QRS_NEXT_CUT()
PTP {E1 28616.845,E2 28616.845}
PTP {X 0,Y 607.911,A -85,B 0,C 180,E1 28616.845,E2 28616.845,E3 0,E4 0,E5 0,E6 0}
QRS_SPEED_INIT()
LIN {X 0,Y 607.911,Z 1007,A -85,B 0,C 180,E1 28616.845,E2 28616.845,E3 0,E4 0,E5 0,E6 0} C_VEL
LIN {X 0,Y 607.911,Z 513.151,A -85,B 0,C 180,E1 28616.845,E2 28616.845} C_VEL
LIN {X 0,Y 607.911,Z 505.074,A -85,B 0,C 180,E1 28616.845,E2 28616.845} C_VEL
LIN {X 0,Y 607.884,Z 503.074,A -85,B 0,C 180,E1 28616.656,E2 28616.656} C_VEL
LIN {X 0,Y 607.844,Z 503.075,A -85,B 0,C 180,E1 28613.767,E2 28613.767} C_VEL
LIN {X 0,Y 607.909,Z 503.072,A -85,B 0,C 180,E1 28610.629,E2 28610.629} C_VEL
LIN {X 0,Y 607.85,Z 503.075,A -85,B 0,C 180,E1 28607.652,E2 28607.652} C_VEL
LIN {X 0,Y 607.919,Z 503.071,A -85,B 0,C 180,E1 28604.516,E2 28604.516} C_VEL
LIN {X 0,Y 607.857,Z 503.074,A -85,B 0,C 180,E1 28601.49,E2 28601.49} C_VEL
LIN {X 0,Y 607.914,Z 503.072,A -85,B 0,C 180,E1 28598.381,E2 28598.381} C_VEL
LIN {X 0,Y 607.861,Z 503.073,A -85,B 0,C 180,E1 28595.408,E2 28595.408} C_VEL
LIN {X 0,Y 607.914,Z 503.074,A -85,B 0,C 180,E1 28592.366,E2 28592.366} C_VEL
LIN {X 0,Y 607.868,Z 503.073,A -85,B 0,C 180,E1 28589.232,E2 28589.232} C_VEL
LIN {X 0,Y 607.912,Z 503.072,A -85,B 0,C 180,E1 28586.112,E2 28586.112} C_VEL
LIN {X 0,Y 607.875,Z 503.073,A -85,B 0,C 180,E1 28582.985,E2 28582.985} C_VEL
LIN {X 0,Y 607.911,Z 503.07,A -85,B 0,C 180,E1 28579.853,E2 28579.853} C_VEL
LIN {X 0,Y 607.88,Z 503.075,A -85,B 0,C 180,E1 28576.767,E2 28576.767} C_VEL
LIN {X 0,Y 607.909,Z 503.417,A -85,B 0,C 180,E1 28576.324,E2 28576.324} C_VEL
LIN {X 0,Y 607.911,Z 532.423,A -85,B 0,C 180,E1 28573.229,E2 28573.229} C_VEL
LIN {X 0,Y 607.861,Z 561.577,A -85,B 0,C 180,E1 28570.197,E2 28570.197} C_VEL
LIN {X 0,Y 607.901,Z 593.601,A -85,B 0,C 180,E1 28566.93,E2 28566.93} C_VEL
LIN {X 0,Y 607.866,Z 623.977,A -85,B 0,C 180,E1 28563.886,E2 28563.886} C_VEL
LIN {X 0,Y 607.91,Z 633.18,A -85,B 0,C 180,E1 28563.011,E2 28563.011} C_VEL
LIN {X 0,Y 607.879,Z 744.156,A -85,B 0,C 180,E1 28561.669,E2 28561.669} C_VEL
LIN {X 0,Y 607.913,Z 759.228,A -85,B 0,C 180,E1 28561.31,E2 28561.31} C_VEL
LIN {X 0,Y 607.919,Z 774.015,A -85,B 0,C 180,E1 28560.76,E2 28560.76} C_VEL
LIN {X 0,Y 607.887,Z 786.969,A -85,B 0,C 180,E1 28560.097,E2 28560.097} C_VEL
LIN {X 0,Y 607.92,Z 799.139,A -85,B 0,C 180,E1 28559.289,E2 28559.289} C_VEL
LIN {X 0,Y 607.919,Z 809.968,A -85,B 0,C 180,E1 28558.366,E2 28558.366} C_VEL
LIN {X 0,Y 607.917,Z 819.55,A -85,B 0,C 180,E1 28557.357,E2 28557.357} C_VEL
LIN {X 0,Y 607.917,Z 828.81,A -85,B 0,C 180,E1 28556.1,E2 28556.1} C_VEL
LIN {X 0,Y 607.917,Z 836.072,A -85,B 0,C 180,E1 28554.784,E2 28554.784} C_VEL
LIN {X 0,Y 607.916,Z 841.374,A -85,B 0,C 180,E1 28553.451,E2 28553.451} C_VEL
LIN {X 0,Y 607.917,Z 845.07,A -85,B 0,C 180,E1 28552.021,E2 28552.021} C_VEL
LIN {X 0,Y 607.918,Z 846.862,A -85,B 0,C 180,E1 28550.504,E2 28550.504} C_VEL
LIN {X 0,Y 607.914,Z 846.58,A -85,B 0,C 180,E1 28549.002,E2 28549.002} C_VEL
LIN {X 0,Y 607.914,Z 844.49,A -85,B 0,C 180,E1 28547.613,E2 28547.613} C_VEL
LIN {X 0,Y 607.915,Z 840.63,A -85,B 0,C 180,E1 28546.234,E2 28546.234} C_VEL
LIN {X 0,Y 607.915,Z 834.801,A -85,B 0,C 180,E1 28544.865,E2 28544.865} C_VEL
LIN {X 0,Y 607.915,Z 827.41,A -85,B 0,C 180,E1 28543.601,E2 28543.601} C_VEL
LIN {X 0,Y 607.919,Z 818.592,A -85,B 0,C 180,E1 28542.44,E2 28542.44} C_VEL
LIN {X 0,Y 607.918,Z 807.23,A -85,B 0,C 180,E1 28541.285,E2 28541.285} C_VEL
LIN {X 0,Y 607.915,Z 795.047,A -85,B 0,C 180,E1 28540.326,E2 28540.326} C_VEL
LIN {X 0,Y 607.906,Z 781.548,A -85,B 0,C 180,E1 28539.513,E2 28539.513} C_VEL
LIN {X 0,Y 607.917,Z 767.716,A -85,B 0,C 180,E1 28538.892,E2 28538.892} C_VEL
LIN {X 0,Y 607.918,Z 753.447,A -85,B 0,C 180,E1 28538.439,E2 28538.439} C_VEL
LIN {X 0,Y 607.905,Z 737.614,A -85,B 0,C 180,E1 28538.142,E2 28538.142} C_VEL
LIN {X 0,Y 607.918,Z 633.091,A -85,B 0,C 180,E1 28536.894,E2 28536.894} C_VEL
LIN {X 0,Y 607.891,Z 611.812,A -85,B 0,C 180,E1 28534.81,E2 28534.81} C_VEL
LIN {X 0,Y 607.883,Z 580.938,A -85,B 0,C 180,E1 28531.695,E2 28531.695} C_VEL
LIN {X 0,Y 607.916,Z 551.557,A -85,B 0,C 180,E1 28528.68,E2 28528.68} C_VEL
LIN {X 0,Y 607.916,Z 520.967,A -85,B 0,C 180,E1 28525.471,E2 28525.471} C_VEL
LIN {X 0,Y 607.9,Z 503.204,A -85,B 0,C 180,E1 28523.542,E2 28523.542} C_VEL
LIN {X 0,Y 607.833,Z 503.077,A -85,B 0,C 180,E1 28520.627,E2 28520.627} C_VEL
LIN {X 0,Y 607.908,Z 503.075,A -85,B 0,C 180,E1 28517.654,E2 28517.654} C_VEL
LIN {X 0,Y 607.83,Z 503.077,A -85,B 0,C 180,E1 28514.545,E2 28514.545} C_VEL
LIN {X 0,Y 607.871,Z 503.076,A -85,B 0,C 180,E1 28511.69,E2 28511.69} C_VEL
LIN {X 0,Y 607.837,Z 503.077,A -85,B 0,C 180,E1 28508.582,E2 28508.582} C_VEL
LIN {X 0,Y 607.837,Z 503.076,A -85,B 0,C 180,E1 28505.822,E2 28505.822} C_VEL
LIN {X 0,Y 607.848,Z 503.077,A -85,B 0,C 180,E1 28502.577,E2 28502.577} C_VEL
LIN {X 0,Y 607.826,Z 503.076,A -85,B 0,C 180,E1 28499.779,E2 28499.779} C_VEL
LIN {X 0,Y 607.882,Z 503.077,A -85,B 0,C 180,E1 28496.676,E2 28496.676} C_VEL
LIN {X 0,Y 607.824,Z 503.077,A -85,B 0,C 180,E1 28493.806,E2 28493.806} C_VEL
LIN {X 0,Y 607.913,Z 503.078,A -85,B 0,C 180,E1 28490.714,E2 28490.714} C_VEL
LIN {X 0,Y 607.828,Z 503.076,A -85,B 0,C 180,E1 28487.72,E2 28487.72} C_VEL
LIN {X 0,Y 607.858,Z 503.077,A -85,B 0,C 180,E1 28484.988,E2 28484.988} C_VEL
LIN {X 0,Y 607.841,Z 503.076,A -85,B 0,C 180,E1 28481.775,E2 28481.775} C_VEL
LIN {X 0,Y 607.841,Z 503.076,A -85,B 0,C 180,E1 28479.051,E2 28479.051} C_VEL
LIN {X 0,Y 607.864,Z 503.075,A -85,B 0,C 180,E1 28475.819,E2 28475.819} C_VEL
LIN {X 0,Y 607.835,Z 503.076,A -85,B 0,C 180,E1 28473.102,E2 28473.102} C_VEL
LIN {X 0,Y 607.918,Z 503.074,A -85,B 0,C 180,E1 28470,E2 28470} C_VEL
LIN {X 0,Y 607.837,Z 503.075,A -85,B 0,C 180,E1 28467.001,E2 28467.001} C_VEL
LIN {X 0,Y 607.917,Z 503.077,A -85,B 0,C 180,E1 28463.97,E2 28463.97} C_VEL
LIN {X 0,Y 607.841,Z 503.075,A -85,B 0,C 180,E1 28460.891,E2 28460.891} C_VEL
LIN {X 0,Y 607.904,Z 503.077,A -85,B 0,C 180,E1 28457.913,E2 28457.913} C_VEL
LIN {X 0,Y 607.85,Z 503.074,A -85,B 0,C 180,E1 28454.869,E2 28454.869} C_VEL
LIN {X 0,Y 607.876,Z 503.076,A -85,B 0,C 180,E1 28451.961,E2 28451.961} C_VEL
LIN {X 0,Y 607.86,Z 503.073,A -85,B 0,C 180,E1 28448.8,E2 28448.8} C_VEL
LIN {X 0,Y 607.863,Z 503.076,A -85,B 0,C 180,E1 28445.948,E2 28445.948} C_VEL
LIN {X 0,Y 607.865,Z 503.073,A -85,B 0,C 180,E1 28442.64,E2 28442.64} C_VEL
LIN {X 0,Y 607.869,Z 503.075,A -85,B 0,C 180,E1 28439.717,E2 28439.717} C_VEL
LIN {X 0,Y 607.865,Z 503.072,A -85,B 0,C 180,E1 28436.417,E2 28436.417} C_VEL
LIN {X 0,Y 607.876,Z 503.076,A -85,B 0,C 180,E1 28433.483,E2 28433.483} C_VEL
LIN {X 0,Y 607.869,Z 503.072,A -85,B 0,C 180,E1 28430.246,E2 28430.246} C_VEL
LIN {X 0,Y 607.883,Z 503.076,A -85,B 0,C 180,E1 28427.242,E2 28427.242} C_VEL
LIN {X 0,Y 607.872,Z 503.071,A -85,B 0,C 180,E1 28424.057,E2 28424.057} C_VEL
LIN {X 0,Y 607.888,Z 503.076,A -85,B 0,C 180,E1 28421.032,E2 28421.032} C_VEL
LIN {X 0,Y 607.868,Z 503.072,A -85,B 0,C 180,E1 28417.771,E2 28417.771} C_VEL
LIN {X 0,Y 607.899,Z 503.077,A -85,B 0,C 180,E1 28414.765,E2 28414.765} C_VEL
LIN {X 0,Y 607.872,Z 503.071,A -85,B 0,C 180,E1 28411.617,E2 28411.617} C_VEL
LIN {X 0,Y 607.902,Z 503.077,A -85,B 0,C 180,E1 28408.574,E2 28408.574} C_VEL
LIN {X 0,Y 607.873,Z 503.071,A -85,B 0,C 180,E1 28405.426,E2 28405.426} C_VEL
LIN {X 0,Y 607.914,Z 503.078,A -85,B 0,C 180,E1 28402.286,E2 28402.286} C_VEL
LIN {X 0,Y 607.871,Z 503.071,A -85,B 0,C 180,E1 28399.107,E2 28399.107} C_VEL
LIN {X 0,Y 607.914,Z 503.075,A -85,B 0,C 180,E1 28395.948,E2 28395.948} C_VEL
LIN {X 0,Y 607.87,Z 503.072,A -85,B 0,C 180,E1 28392.811,E2 28392.811} C_VEL
LIN {X 0,Y 607.914,Z 503.075,A -85,B 0,C 180,E1 28389.774,E2 28389.774} C_VEL
LIN {X 0,Y 607.873,Z 503.072,A -85,B 0,C 180,E1 28386.613,E2 28386.613} C_VEL
LIN {X 0,Y 607.911,Z 503.073,A -85,B 0,C 180,E1 28383.5,E2 28383.5} C_VEL
LIN {X 0,Y 607.875,Z 503.072,A -85,B 0,C 180,E1 28380.437,E2 28380.437} C_VEL
LIN {X 0,Y 607.901,Z 503.299,A -85,B 0,C 180,E1 28379.782,E2 28379.782} C_VEL
LIN {X 0,Y 607.917,Z 514.846,A -85,B 0,C 180,E1 28378.956,E2 28378.956} C_VEL
LIN {X 0,Y 607.891,Z 559.528,A -85,B 0,C 180,E1 28375.944,E2 28375.944} C_VEL
LIN {X 0,Y 607.91,Z 607.569,A -85,B 0,C 180,E1 28372.788,E2 28372.788} C_VEL
LIN {X 0,Y 607.906,Z 615.06,A -85,B 0,C 180,E1 28372.329,E2 28372.329} C_VEL
LIN {X 0,Y 607.912,Z 824.351,A -85,B 0,C 180,E1 28369.704,E2 28369.704} C_VEL
LIN {X 0,Y 607.892,Z 842.612,A -85,B 0,C 180,E1 28369.305,E2 28369.305} C_VEL
LIN {X 0,Y 607.91,Z 860.78,A -85,B 0,C 180,E1 28368.731,E2 28368.731} C_VEL
LIN {X 0,Y 607.886,Z 879.07,A -85,B 0,C 180,E1 28367.963,E2 28367.963} C_VEL
LIN {X 0,Y 607.919,Z 895.797,A -85,B 0,C 180,E1 28367.072,E2 28367.072} C_VEL
LIN {X 0,Y 607.916,Z 911.646,A -85,B 0,C 180,E1 28366.04,E2 28366.04} C_VEL
LIN {X 0,Y 607.917,Z 926.565,A -85,B 0,C 180,E1 28364.867,E2 28364.867} C_VEL
LIN {X 0,Y 607.918,Z 940.218,A -85,B 0,C 180,E1 28363.582,E2 28363.582} C_VEL
LIN {X 0,Y 607.917,Z 952.906,A -85,B 0,C 180,E1 28362.153,E2 28362.153} C_VEL
LIN {X 0,Y 607.913,Z 964.223,A -85,B 0,C 180,E1 28360.615,E2 28360.615} C_VEL
LIN {X 0,Y 607.918,Z 973.987,A -85,B 0,C 180,E1 28358.99,E2 28358.99} C_VEL
LIN {X 0,Y 607.909,Z 981.864,A -85,B 0,C 180,E1 28357.35,E2 28357.35} C_VEL
LIN {X 0,Y 607.906,Z 988.106,A -85,B 0,C 180,E1 28355.664,E2 28355.664} C_VEL
LIN {X 0,Y 607.917,Z 992.871,A -85,B 0,C 180,E1 28353.867,E2 28353.867} C_VEL
LIN {X 0,Y 607.916,Z 995.786,A -85,B 0,C 180,E1 28352.075,E2 28352.075} C_VEL
LIN {X 0,Y 607.907,Z 996.939,A -85,B 0,C 180,E1 28350.284,E2 28350.284} C_VEL
LIN {X 0,Y 607.915,Z 996.349,A -85,B 0,C 180,E1 28348.493,E2 28348.493} C_VEL
LIN {X 0,Y 607.908,Z 994.007,A -85,B 0,C 180,E1 28346.701,E2 28346.701} C_VEL
LIN {X 0,Y 607.905,Z 990.1,A -85,B 0,C 180,E1 28345.001,E2 28345.001} C_VEL
LIN {X 0,Y 607.913,Z 984.473,A -85,B 0,C 180,E1 28343.296,E2 28343.296} C_VEL
LIN {X 0,Y 607.915,Z 977.431,A -85,B 0,C 180,E1 28341.68,E2 28341.68} C_VEL
LIN {X 0,Y 607.91,Z 968.521,A -85,B 0,C 180,E1 28340.057,E2 28340.057} C_VEL
LIN {X 0,Y 607.919,Z 958.16,A -85,B 0,C 180,E1 28338.523,E2 28338.523} C_VEL
LIN {X 0,Y 607.914,Z 946.365,A -85,B 0,C 180,E1 28337.077,E2 28337.077} C_VEL
LIN {X 0,Y 607.916,Z 933.113,A -85,B 0,C 180,E1 28335.72,E2 28335.72} C_VEL
LIN {X 0,Y 607.917,Z 918.266,A -85,B 0,C 180,E1 28334.452,E2 28334.452} C_VEL
LIN {X 0,Y 607.918,Z 902.26,A -85,B 0,C 180,E1 28333.324,E2 28333.324} C_VEL
LIN {X 0,Y 607.895,Z 886.08,A -85,B 0,C 180,E1 28332.386,E2 28332.386} C_VEL
LIN {X 0,Y 607.907,Z 869.132,A -85,B 0,C 180,E1 28331.594,E2 28331.594} C_VEL
LIN {X 0,Y 607.892,Z 850.474,A -85,B 0,C 180,E1 28330.922,E2 28330.922} C_VEL
LIN {X 0,Y 607.901,Z 832.403,A -85,B 0,C 180,E1 28330.451,E2 28330.451} C_VEL
LIN {X 0,Y 607.919,Z 812.939,A -85,B 0,C 180,E1 28330.13,E2 28330.13} C_VEL
LIN {X 0,Y 607.906,Z 614.386,A -85,B 0,C 180,E1 28327.648,E2 28327.648} C_VEL
LIN {X 0,Y 607.907,Z 568.229,A -85,B 0,C 180,E1 28324.634,E2 28324.634} C_VEL
LIN {X 0,Y 607.917,Z 521.763,A -85,B 0,C 180,E1 28321.516,E2 28321.516} C_VEL
LIN {X 0,Y 607.904,Z 503.513,A -85,B 0,C 180,E1 28320.249,E2 28320.249} C_VEL
LIN {X 0,Y 607.883,Z 503.075,A -85,B 0,C 180,E1 28320.003,E2 28320.003} C_VEL
LIN {X 0,Y 607.917,Z 503.068,A -85,B 0,C 180,E1 28316.842,E2 28316.842} C_VEL
LIN {X 0,Y 607.873,Z 503.074,A -85,B 0,C 180,E1 28313.696,E2 28313.696} C_VEL
LIN {X 0,Y 607.915,Z 503.07,A -85,B 0,C 180,E1 28310.595,E2 28310.595} C_VEL
LIN {X 0,Y 607.864,Z 503.074,A -85,B 0,C 180,E1 28307.468,E2 28307.468} C_VEL
LIN {X 0,Y 607.918,Z 503.07,A -85,B 0,C 180,E1 28304.461,E2 28304.461} C_VEL
LIN {X 0,Y 607.858,Z 503.074,A -85,B 0,C 180,E1 28301.268,E2 28301.268} C_VEL
LIN {X 0,Y 607.918,Z 503.072,A -85,B 0,C 180,E1 28298.178,E2 28298.178} C_VEL
LIN {X 0,Y 607.852,Z 503.075,A -85,B 0,C 180,E1 28295.15,E2 28295.15} C_VEL
LIN {X 0,Y 607.91,Z 503.072,A -85,B 0,C 180,E1 28292.118,E2 28292.118} C_VEL
LIN {X 0,Y 607.847,Z 503.075,A -85,B 0,C 180,E1 28289.029,E2 28289.029} C_VEL
LIN {X 0,Y 607.883,Z 503.074,A -85,B 0,C 180,E1 28286.107,E2 28286.107} C_VEL
LIN {X 0,Y 607.842,Z 503.076,A -85,B 0,C 180,E1 28282.918,E2 28282.918} C_VEL
LIN {X 0,Y 607.859,Z 503.075,A -85,B 0,C 180,E1 28280.095,E2 28280.095} C_VEL
LIN {X 0,Y 607.839,Z 503.077,A -85,B 0,C 180,E1 28276.828,E2 28276.828} C_VEL
LIN {X 0,Y 607.833,Z 503.076,A -85,B 0,C 180,E1 28274.188,E2 28274.188} C_VEL
LIN {X 0,Y 607.862,Z 503.077,A -85,B 0,C 180,E1 28271,E2 28271} C_VEL
LIN {X 0,Y 607.825,Z 503.077,A -85,B 0,C 180,E1 28268.228,E2 28268.228} C_VEL
LIN {X 0,Y 607.913,Z 503.077,A -85,B 0,C 180,E1 28265.19,E2 28265.19} C_VEL
LIN {X 0,Y 607.833,Z 503.076,A -85,B 0,C 180,E1 28262.168,E2 28262.168} C_VEL
LIN {X 0,Y 607.909,Z 503.078,A -85,B 0,C 180,E1 28259.152,E2 28259.152} C_VEL
LIN {X 0,Y 607.884,Z 503.074,A -85,B 0,C 180,E1 28256.656,E2 28256.656} C_VEL
LIN {X 0,Y 606.826,Z 503.205,A -85,B 0,C 180,E1 28255.93,E2 28255.93} C_VEL
LIN {X 0,Y 600.415,Z 504.003,A -85,B 0,C 180,E1 28253.894,E2 28253.894} C_VEL
LIN {X 0,Y 599.932,Z 504.065,A -85,B 0,C 180,E1 28253.364,E2 28253.364} C_VEL
LIN {X 0,Y 599.917,Z 504.062,A -85,B 0,C 180,E1 28250.115,E2 28250.115} C_VEL
LIN {X 0,Y 599.939,Z 504.065,A -85,B 0,C 180,E1 28247.193,E2 28247.193} C_VEL
LIN {X 0,Y 599.923,Z 504.062,A -85,B 0,C 180,E1 28243.939,E2 28243.939} C_VEL
LIN {X 0,Y 599.963,Z 504.066,A -85,B 0,C 180,E1 28240.878,E2 28240.878} C_VEL
LIN {X 0,Y 599.924,Z 504.062,A -85,B 0,C 180,E1 28237.651,E2 28237.651} C_VEL
LIN {X 0,Y 599.978,Z 504.065,A -85,B 0,C 180,E1 28234.535,E2 28234.535} C_VEL
LIN {X 0,Y 599.928,Z 504.062,A -85,B 0,C 180,E1 28231.424,E2 28231.424} C_VEL
LIN {X 0,Y 599.976,Z 504.064,A -85,B 0,C 180,E1 28228.335,E2 28228.335} C_VEL
LIN {X 0,Y 599.934,Z 504.061,A -85,B 0,C 180,E1 28225.24,E2 28225.24} C_VEL
LIN {X 0,Y 599.974,Z 504.064,A -85,B 0,C 180,E1 28222.17,E2 28222.17} C_VEL
LIN {X 0,Y 599.939,Z 504.063,A -85,B 0,C 180,E1 28218.955,E2 28218.955} C_VEL
LIN {X 0,Y 599.983,Z 504.317,A -85,B 0,C 180,E1 28216.609,E2 28216.609} C_VEL
LIN {X 0,Y 600.305,Z 508.323,A -85,B 0,C 180,E1 28216.141,E2 28216.141} C_VEL
LIN {X 0,Y 600.213,Z 538.089,A -85,B 0,C 180,E1 28212.941,E2 28212.941} C_VEL
LIN {X 0,Y 600.13,Z 568.295,A -85,B 0,C 180,E1 28209.769,E2 28209.769} C_VEL
LIN {X 0,Y 600.067,Z 599.365,A -85,B 0,C 180,E1 28206.569,E2 28206.569} C_VEL
LIN {X 0,Y 600.003,Z 631.076,A -85,B 0,C 180,E1 28203.357,E2 28203.357} C_VEL
LIN {X 0,Y 600.096,Z 633.638,A -85,B 0,C 180,E1 28203.176,E2 28203.176} C_VEL
LIN {X 0,Y 600.042,Z 744.434,A -85,B 0,C 180,E1 28201.819,E2 28201.819} C_VEL
LIN {X 0,Y 600.058,Z 759.369,A -85,B 0,C 180,E1 28201.456,E2 28201.456} C_VEL
LIN {X 0,Y 600.039,Z 774.355,A -85,B 0,C 180,E1 28200.889,E2 28200.889} C_VEL
LIN {X 0,Y 599.979,Z 787.292,A -85,B 0,C 180,E1 28200.213,E2 28200.213} C_VEL
LIN {X 0,Y 599.985,Z 799.854,A -85,B 0,C 180,E1 28199.358,E2 28199.358} C_VEL
LIN {X 0,Y 599.962,Z 810.146,A -85,B 0,C 180,E1 28198.461,E2 28198.461} C_VEL
LIN {X 0,Y 599.943,Z 819.714,A -85,B 0,C 180,E1 28197.436,E2 28197.436} C_VEL
LIN {X 0,Y 599.931,Z 828.658,A -85,B 0,C 180,E1 28196.206,E2 28196.206} C_VEL
LIN {X 0,Y 599.923,Z 835.651,A -85,B 0,C 180,E1 28194.936,E2 28194.936} C_VEL
LIN {X 0,Y 599.92,Z 840.797,A -85,B 0,C 180,E1 28193.679,E2 28193.679} C_VEL
LIN {X 0,Y 599.916,Z 844.706,A -85,B 0,C 180,E1 28192.227,E2 28192.227} C_VEL
LIN {X 0,Y 599.915,Z 846.599,A -85,B 0,C 180,E1 28190.892,E2 28190.892} C_VEL
LIN {X 0,Y 599.915,Z 846.893,A -85,B 0,C 180,E1 28189.468,E2 28189.468} C_VEL
LIN {X 0,Y 599.917,Z 845.391,A -85,B 0,C 180,E1 28188.056,E2 28188.056} C_VEL
LIN {X 0,Y 599.917,Z 842.141,A -85,B 0,C 180,E1 28186.656,E2 28186.656} C_VEL
LIN {X 0,Y 599.92,Z 836.744,A -85,B 0,C 180,E1 28185.204,E2 28185.204} C_VEL
LIN {X 0,Y 599.929,Z 829.752,A -85,B 0,C 180,E1 28183.884,E2 28183.884} C_VEL
LIN {X 0,Y 599.942,Z 821.575,A -85,B 0,C 180,E1 28182.706,E2 28182.706} C_VEL
LIN {X 0,Y 599.958,Z 812.955,A -85,B 0,C 180,E1 28181.729,E2 28181.729} C_VEL
LIN {X 0,Y 599.979,Z 802.998,A -85,B 0,C 180,E1 28180.804,E2 28180.804} C_VEL
LIN {X 0,Y 599.984,Z 790.324,A -85,B 0,C 180,E1 28179.882,E2 28179.882} C_VEL
LIN {X 0,Y 600.029,Z 777.198,A -85,B 0,C 180,E1 28179.155,E2 28179.155} C_VEL
LIN {X 0,Y 600.057,Z 763.751,A -85,B 0,C 180,E1 28178.598,E2 28178.598} C_VEL
LIN {X 0,Y 600.076,Z 748.239,A -85,B 0,C 180,E1 28178.164,E2 28178.164} C_VEL
LIN {X 0,Y 600.068,Z 729.544,A -85,B 0,C 180,E1 28177.887,E2 28177.887} C_VEL
LIN {X 0,Y 600.054,Z 633.14,A -85,B 0,C 180,E1 28176.723,E2 28176.723} C_VEL
LIN {X 0,Y 600.026,Z 620.12,A -85,B 0,C 180,E1 28175.449,E2 28175.449} C_VEL
LIN {X 0,Y 600.054,Z 590.046,A -85,B 0,C 180,E1 28172.386,E2 28172.386} C_VEL
LIN {X 0,Y 600.127,Z 559.615,A -85,B 0,C 180,E1 28169.235,E2 28169.235} C_VEL
LIN {X 0,Y 600.211,Z 530.678,A -85,B 0,C 180,E1 28166.178,E2 28166.178} C_VEL
LIN {X 0,Y 600.23,Z 505.406,A -85,B 0,C 180,E1 28163.447,E2 28163.447} C_VEL
LIN {X 0,Y 599.936,Z 504.157,A -85,B 0,C 180,E1 28163.252,E2 28163.252} C_VEL
LIN {X 0,Y 599.898,Z 504.066,A -85,B 0,C 180,E1 28160.405,E2 28160.405} C_VEL
LIN {X 0,Y 599.949,Z 504.066,A -85,B 0,C 180,E1 28157.292,E2 28157.292} C_VEL
LIN {X 0,Y 599.891,Z 504.066,A -85,B 0,C 180,E1 28154.335,E2 28154.335} C_VEL
LIN {X 0,Y 599.967,Z 504.066,A -85,B 0,C 180,E1 28151.238,E2 28151.238} C_VEL
LIN {X 0,Y 599.888,Z 504.066,A -85,B 0,C 180,E1 28148.284,E2 28148.284} C_VEL
LIN {X 0,Y 599.958,Z 504.063,A -85,B 0,C 180,E1 28145.268,E2 28145.268} C_VEL
LIN {X 0,Y 599.886,Z 504.066,A -85,B 0,C 180,E1 28142.182,E2 28142.182} C_VEL
LIN {X 0,Y 599.937,Z 504.064,A -85,B 0,C 180,E1 28139.228,E2 28139.228} C_VEL
LIN {X 0,Y 599.887,Z 504.066,A -85,B 0,C 180,E1 28136.06,E2 28136.06} C_VEL
LIN {X 0,Y 599.914,Z 504.066,A -85,B 0,C 180,E1 28133.252,E2 28133.252} C_VEL
LIN {X 0,Y 599.901,Z 504.066,A -85,B 0,C 180,E1 28130.058,E2 28130.058} C_VEL
LIN {X 0,Y 599.898,Z 504.065,A -85,B 0,C 180,E1 28127.288,E2 28127.288} C_VEL
LIN {X 0,Y 599.915,Z 504.065,A -85,B 0,C 180,E1 28124.028,E2 28124.028} C_VEL
LIN {X 0,Y 599.898,Z 504.064,A -85,B 0,C 180,E1 28121.175,E2 28121.175} C_VEL
LIN {X 0,Y 599.935,Z 504.064,A -85,B 0,C 180,E1 28117.977,E2 28117.977} C_VEL
LIN {X 0,Y 599.897,Z 504.064,A -85,B 0,C 180,E1 28115.084,E2 28115.084} C_VEL
LIN {X 0,Y 599.966,Z 504.063,A -85,B 0,C 180,E1 28111.983,E2 28111.983} C_VEL
LIN {X 0,Y 599.898,Z 504.065,A -85,B 0,C 180,E1 28108.959,E2 28108.959} C_VEL
LIN {X 0,Y 599.975,Z 504.062,A -85,B 0,C 180,E1 28105.861,E2 28105.861} C_VEL
LIN {X 0,Y 599.901,Z 504.064,A -85,B 0,C 180,E1 28102.835,E2 28102.835} C_VEL
LIN {X 0,Y 599.978,Z 504.063,A -85,B 0,C 180,E1 28099.773,E2 28099.773} C_VEL
LIN {X 0,Y 599.904,Z 504.062,A -85,B 0,C 180,E1 28096.759,E2 28096.759} C_VEL
LIN {X 0,Y 599.966,Z 504.066,A -85,B 0,C 180,E1 28093.787,E2 28093.787} C_VEL
LIN {X 0,Y 599.909,Z 504.062,A -85,B 0,C 180,E1 28090.661,E2 28090.661} C_VEL
LIN {X 0,Y 599.958,Z 504.064,A -85,B 0,C 180,E1 28087.662,E2 28087.662} C_VEL
LIN {X 0,Y 599.913,Z 504.063,A -85,B 0,C 180,E1 28084.493,E2 28084.493} C_VEL
LIN {X 0,Y 599.955,Z 504.065,A -85,B 0,C 180,E1 28081.528,E2 28081.528} C_VEL
LIN {X 0,Y 599.919,Z 504.062,A -85,B 0,C 180,E1 28078.377,E2 28078.377} C_VEL
LIN {X 0,Y 599.948,Z 504.066,A -85,B 0,C 180,E1 28075.412,E2 28075.412} C_VEL
LIN {X 0,Y 599.925,Z 504.06,A -85,B 0,C 180,E1 28072.242,E2 28072.242} C_VEL
LIN {X 0,Y 599.95,Z 504.065,A -85,B 0,C 180,E1 28069.242,E2 28069.242} C_VEL
LIN {X 0,Y 599.926,Z 504.06,A -85,B 0,C 180,E1 28066.015,E2 28066.015} C_VEL
LIN {X 0,Y 599.954,Z 504.065,A -85,B 0,C 180,E1 28063.043,E2 28063.043} C_VEL
LIN {X 0,Y 599.928,Z 504.06,A -85,B 0,C 180,E1 28059.819,E2 28059.819} C_VEL
LIN {X 0,Y 599.978,Z 504.066,A -85,B 0,C 180,E1 28056.661,E2 28056.661} C_VEL
LIN {X 0,Y 599.925,Z 504.06,A -85,B 0,C 180,E1 28053.471,E2 28053.471} C_VEL
LIN {X 0,Y 599.979,Z 504.065,A -85,B 0,C 180,E1 28050.441,E2 28050.441} C_VEL
LIN {X 0,Y 599.928,Z 504.061,A -85,B 0,C 180,E1 28047.309,E2 28047.309} C_VEL
LIN {X 0,Y 599.977,Z 504.064,A -85,B 0,C 180,E1 28044.201,E2 28044.201} C_VEL
LIN {X 0,Y 599.929,Z 504.061,A -85,B 0,C 180,E1 28041.074,E2 28041.074} C_VEL
LIN {X 0,Y 599.974,Z 504.063,A -85,B 0,C 180,E1 28037.938,E2 28037.938} C_VEL
LIN {X 0,Y 599.931,Z 504.061,A -85,B 0,C 180,E1 28034.825,E2 28034.825} C_VEL
LIN {X 0,Y 599.973,Z 504.062,A -85,B 0,C 180,E1 28031.704,E2 28031.704} C_VEL
LIN {X 0,Y 599.933,Z 504.062,A -85,B 0,C 180,E1 28028.556,E2 28028.556} C_VEL
LIN {X 0,Y 599.973,Z 504.061,A -85,B 0,C 180,E1 28025.42,E2 28025.42} C_VEL
LIN {X 0,Y 599.937,Z 504.061,A -85,B 0,C 180,E1 28022.228,E2 28022.228} C_VEL
LIN {X 0,Y 599.972,Z 504.303,A -85,B 0,C 180,E1 28020.143,E2 28020.143} C_VEL
LIN {X 0,Y 600.653,Z 507.548,A -85,B 0,C 180,E1 28019.848,E2 28019.848} C_VEL
LIN {X 0,Y 600.489,Z 551.772,A -85,B 0,C 180,E1 28016.814,E2 28016.814} C_VEL
LIN {X 0,Y 600.375,Z 597.331,A -85,B 0,C 180,E1 28013.766,E2 28013.766} C_VEL
LIN {X 0,Y 600.405,Z 615.06,A -85,B 0,C 180,E1 28012.623,E2 28012.623} C_VEL
LIN {X 0,Y 600.372,Z 824.351,A -85,B 0,C 180,E1 28009.962,E2 28009.962} C_VEL
LIN {X 0,Y 600.312,Z 843.223,A -85,B 0,C 180,E1 28009.541,E2 28009.541} C_VEL
LIN {X 0,Y 600.281,Z 861.422,A -85,B 0,C 180,E1 28008.953,E2 28008.953} C_VEL
LIN {X 0,Y 600.204,Z 879.067,A -85,B 0,C 180,E1 28008.2,E2 28008.2} C_VEL
LIN {X 0,Y 600.179,Z 895.713,A -85,B 0,C 180,E1 28007.304,E2 28007.304} C_VEL
LIN {X 0,Y 600.122,Z 911.645,A -85,B 0,C 180,E1 28006.254,E2 28006.254} C_VEL
LIN {X 0,Y 600.069,Z 926.566,A -85,B 0,C 180,E1 28005.066,E2 28005.066} C_VEL
LIN {X 0,Y 600.02,Z 940.02,A -85,B 0,C 180,E1 28003.786,E2 28003.786} C_VEL
LIN {X 0,Y 599.985,Z 952.907,A -85,B 0,C 180,E1 28002.316,E2 28002.316} C_VEL
LIN {X 0,Y 599.954,Z 964.224,A -85,B 0,C 180,E1 28000.758,E2 28000.758} C_VEL
LIN {X 0,Y 599.934,Z 973.988,A -85,B 0,C 180,E1 27999.11,E2 27999.11} C_VEL
LIN {X 0,Y 599.92,Z 982.043,A -85,B 0,C 180,E1 27997.405,E2 27997.405} C_VEL
LIN {X 0,Y 599.911,Z 988.408,A -85,B 0,C 180,E1 27995.644,E2 27995.644} C_VEL
LIN {X 0,Y 599.918,Z 992.871,A -85,B 0,C 180,E1 27993.919,E2 27993.919} C_VEL
LIN {X 0,Y 599.917,Z 995.786,A -85,B 0,C 180,E1 27992.102,E2 27992.102} C_VEL
LIN {X 0,Y 599.907,Z 996.939,A -85,B 0,C 180,E1 27990.288,E2 27990.288} C_VEL
LIN {X 0,Y 599.915,Z 996.349,A -85,B 0,C 180,E1 27988.473,E2 27988.473} C_VEL
LIN {X 0,Y 599.907,Z 994.008,A -85,B 0,C 180,E1 27986.657,E2 27986.657} C_VEL
LIN {X 0,Y 599.908,Z 990.101,A -85,B 0,C 180,E1 27984.934,E2 27984.934} C_VEL
LIN {X 0,Y 599.92,Z 984.474,A -85,B 0,C 180,E1 27983.206,E2 27983.206} C_VEL
LIN {X 0,Y 599.928,Z 977.432,A -85,B 0,C 180,E1 27981.568,E2 27981.568} C_VEL
LIN {X 0,Y 599.942,Z 968.522,A -85,B 0,C 180,E1 27979.924,E2 27979.924} C_VEL
LIN {X 0,Y 599.969,Z 958.161,A -85,B 0,C 180,E1 27978.369,E2 27978.369} C_VEL
LIN {X 0,Y 600.001,Z 946.366,A -85,B 0,C 180,E1 27976.903,E2 27976.903} C_VEL
LIN {X 0,Y 600.049,Z 932.752,A -85,B 0,C 180,E1 27975.493,E2 27975.493} C_VEL
LIN {X 0,Y 600.103,Z 918.265,A -85,B 0,C 180,E1 27974.244,E2 27974.244} C_VEL
LIN {X 0,Y 600.164,Z 902.263,A -85,B 0,C 180,E1 27973.102,E2 27973.102} C_VEL
LIN {X 0,Y 600.195,Z 885.088,A -85,B 0,C 180,E1 27972.103,E2 27972.103} C_VEL
LIN {X 0,Y 600.277,Z 867.704,A -85,B 0,C 180,E1 27971.295,E2 27971.295} C_VEL
LIN {X 0,Y 600.302,Z 849.613,A -85,B 0,C 180,E1 27970.646,E2 27970.646} C_VEL
LIN {X 0,Y 600.354,Z 831.296,A -85,B 0,C 180,E1 27970.173,E2 27970.173} C_VEL
LIN {X 0,Y 600.395,Z 811.501,A -85,B 0,C 180,E1 27969.852,E2 27969.852} C_VEL
LIN {X 0,Y 600.379,Z 614.841,A -85,B 0,C 180,E1 27967.371,E2 27967.371} C_VEL
LIN {X 0,Y 600.463,Z 568.229,A -85,B 0,C 180,E1 27964.297,E2 27964.297} C_VEL
LIN {X 0,Y 600.607,Z 521.554,A -85,B 0,C 180,E1 27961.123,E2 27961.123} C_VEL
LIN {X 0,Y 600.44,Z 506.011,A -85,B 0,C 180,E1 27960.033,E2 27960.033} C_VEL
LIN {X 0,Y 599.951,Z 504.171,A -85,B 0,C 180,E1 27959.816,E2 27959.816} C_VEL
LIN {X 0,Y 599.975,Z 504.059,A -85,B 0,C 180,E1 27956.756,E2 27956.756} C_VEL
LIN {X 0,Y 599.932,Z 504.063,A -85,B 0,C 180,E1 27953.608,E2 27953.608} C_VEL
LIN {X 0,Y 599.975,Z 504.061,A -85,B 0,C 180,E1 27950.467,E2 27950.467} C_VEL
LIN {X 0,Y 599.925,Z 504.063,A -85,B 0,C 180,E1 27947.423,E2 27947.423} C_VEL
LIN {X 0,Y 599.977,Z 504.06,A -85,B 0,C 180,E1 27944.37,E2 27944.37} C_VEL
LIN {X 0,Y 599.92,Z 504.063,A -85,B 0,C 180,E1 27941.273,E2 27941.273} C_VEL
LIN {X 0,Y 599.978,Z 504.061,A -85,B 0,C 180,E1 27938.141,E2 27938.141} C_VEL
LIN {X 0,Y 599.912,Z 504.063,A -85,B 0,C 180,E1 27935.09,E2 27935.09} C_VEL
LIN {X 0,Y 599.979,Z 504.062,A -85,B 0,C 180,E1 27931.989,E2 27931.989} C_VEL
LIN {X 0,Y 599.905,Z 504.064,A -85,B 0,C 180,E1 27928.904,E2 27928.904} C_VEL
LIN {X 0,Y 599.973,Z 504.063,A -85,B 0,C 180,E1 27925.866,E2 27925.866} C_VEL
LIN {X 0,Y 599.901,Z 504.065,A -85,B 0,C 180,E1 27922.841,E2 27922.841} C_VEL
LIN {X 0,Y 599.934,Z 504.064,A -85,B 0,C 180,E1 27919.97,E2 27919.97} C_VEL
LIN {X 0,Y 599.902,Z 504.066,A -85,B 0,C 180,E1 27916.858,E2 27916.858} C_VEL
LIN {X 0,Y 599.894,Z 504.065,A -85,B 0,C 180,E1 27914.182,E2 27914.182} C_VEL
LIN {X 0,Y 599.918,Z 504.066,A -85,B 0,C 180,E1 27910.953,E2 27910.953} C_VEL
LIN {X 0,Y 599.889,Z 504.066,A -85,B 0,C 180,E1 27908.136,E2 27908.136} C_VEL
LIN {X 0,Y 599.96,Z 504.064,A -85,B 0,C 180,E1 27905.067,E2 27905.067} C_VEL
LIN {X 0,Y 599.894,Z 504.065,A -85,B 0,C 180,E1 27902.101,E2 27902.101} C_VEL
LIN {X 0,Y 599.978,Z 504.065,A -85,B 0,C 180,E1 27899.045,E2 27899.045} C_VEL
LIN {X 0,Y 599.901,Z 504.064,A -85,B 0,C 180,E1 27895.986,E2 27895.986} C_VEL
LIN {X 0,Y 599.932,Z 504.065,A -85,B 0,C 180,E1 27893.364,E2 27893.364} C_VEL
LIN {X 0,Y 598.995,Z 504.189,A -85,B 0,C 180,E1 27892.628,E2 27892.628} C_VEL
LIN {X 0,Y 592.431,Z 504.999,A -85,B 0,C 180,E1 27890.511,E2 27890.511} C_VEL
LIN {X 0,Y 591.974,Z 505.051,A -85,B 0,C 180,E1 27890.026,E2 27890.026} C_VEL
LIN {X 0,Y 592.021,Z 505.055,A -85,B 0,C 180,E1 27887.003,E2 27887.003} C_VEL
LIN {X 0,Y 591.979,Z 505.051,A -85,B 0,C 180,E1 27883.818,E2 27883.818} C_VEL
LIN {X 0,Y 592.036,Z 505.055,A -85,B 0,C 180,E1 27880.728,E2 27880.728} C_VEL
LIN {X 0,Y 591.983,Z 505.051,A -85,B 0,C 180,E1 27877.56,E2 27877.56} C_VEL
LIN {X 0,Y 592.039,Z 505.053,A -85,B 0,C 180,E1 27874.491,E2 27874.491} C_VEL
LIN {X 0,Y 591.989,Z 505.051,A -85,B 0,C 180,E1 27871.336,E2 27871.336} C_VEL
LIN {X 0,Y 592.036,Z 505.051,A -85,B 0,C 180,E1 27868.202,E2 27868.202} C_VEL
LIN {X 0,Y 591.995,Z 505.052,A -85,B 0,C 180,E1 27865.071,E2 27865.071} C_VEL
LIN {X 0,Y 592.038,Z 505.048,A -85,B 0,C 180,E1 27861.821,E2 27861.821} C_VEL
LIN {X 0,Y 592.015,Z 505.056,A -85,B 0,C 180,E1 27858.572,E2 27858.572} C_VEL
LIN {X 0,Y 592.024,Z 505.217,A -85,B 0,C 180,E1 27856.91,E2 27856.91} C_VEL
LIN {X 0,Y 592.705,Z 508.892,A -85,B 0,C 180,E1 27856.44,E2 27856.44} C_VEL
LIN {X 0,Y 592.527,Z 538.628,A -85,B 0,C 180,E1 27853.199,E2 27853.199} C_VEL
LIN {X 0,Y 592.354,Z 568.506,A -85,B 0,C 180,E1 27850.018,E2 27850.018} C_VEL
LIN {X 0,Y 592.228,Z 599.151,A -85,B 0,C 180,E1 27846.818,E2 27846.818} C_VEL
LIN {X 0,Y 592.096,Z 629.625,A -85,B 0,C 180,E1 27843.687,E2 27843.687} C_VEL
LIN {X 0,Y 592.196,Z 633.411,A -85,B 0,C 180,E1 27843.359,E2 27843.359} C_VEL
LIN {X 0,Y 592.209,Z 744.492,A -85,B 0,C 180,E1 27841.977,E2 27841.977} C_VEL
LIN {X 0,Y 592.209,Z 758.628,A -85,B 0,C 180,E1 27841.634,E2 27841.634} C_VEL
LIN {X 0,Y 592.165,Z 772.791,A -85,B 0,C 180,E1 27841.105,E2 27841.105} C_VEL
LIN {X 0,Y 592.086,Z 785.933,A -85,B 0,C 180,E1 27840.434,E2 27840.434} C_VEL
LIN {X 0,Y 592.052,Z 799.13,A -85,B 0,C 180,E1 27839.542,E2 27839.542} C_VEL
LIN {X 0,Y 592.006,Z 810.435,A -85,B 0,C 180,E1 27838.549,E2 27838.549} C_VEL
LIN {X 0,Y 591.972,Z 819.747,A -85,B 0,C 180,E1 27837.533,E2 27837.533} C_VEL
LIN {X 0,Y 591.945,Z 828.833,A -85,B 0,C 180,E1 27836.263,E2 27836.263} C_VEL
LIN {X 0,Y 591.928,Z 836.287,A -85,B 0,C 180,E1 27834.869,E2 27834.869} C_VEL
LIN {X 0,Y 591.919,Z 841.548,A -85,B 0,C 180,E1 27833.49,E2 27833.49} C_VEL
LIN {X 0,Y 591.918,Z 844.981,A -85,B 0,C 180,E1 27832.125,E2 27832.125} C_VEL
LIN {X 0,Y 591.919,Z 846.781,A -85,B 0,C 180,E1 27830.64,E2 27830.64} C_VEL
LIN {X 0,Y 591.916,Z 846.746,A -85,B 0,C 180,E1 27829.219,E2 27829.219} C_VEL
LIN {X 0,Y 591.917,Z 845.01,A -85,B 0,C 180,E1 27827.8,E2 27827.8} C_VEL
LIN {X 0,Y 591.919,Z 841.394,A -85,B 0,C 180,E1 27826.37,E2 27826.37} C_VEL
LIN {X 0,Y 591.929,Z 836.448,A -85,B 0,C 180,E1 27825.075,E2 27825.075} C_VEL
LIN {X 0,Y 591.943,Z 829.01,A -85,B 0,C 180,E1 27823.676,E2 27823.676} C_VEL
LIN {X 0,Y 591.97,Z 820.588,A -85,B 0,C 180,E1 27822.483,E2 27822.483} C_VEL
LIN {X 0,Y 592.002,Z 811.741,A -85,B 0,C 180,E1 27821.494,E2 27821.494} C_VEL
LIN {X 0,Y 592.045,Z 801.479,A -85,B 0,C 180,E1 27820.556,E2 27820.556} C_VEL
LIN {X 0,Y 592.079,Z 789.132,A -85,B 0,C 180,E1 27819.671,E2 27819.671} C_VEL
LIN {X 0,Y 592.156,Z 775.68,A -85,B 0,C 180,E1 27818.935,E2 27818.935} C_VEL
LIN {X 0,Y 592.202,Z 762.127,A -85,B 0,C 180,E1 27818.391,E2 27818.391} C_VEL
LIN {X 0,Y 592.241,Z 747.417,A -85,B 0,C 180,E1 27817.989,E2 27817.989} C_VEL
LIN {X 0,Y 592.243,Z 725.649,A -85,B 0,C 180,E1 27817.678,E2 27817.678} C_VEL
LIN {X 0,Y 592.165,Z 633.126,A -85,B 0,C 180,E1 27816.543,E2 27816.543} C_VEL
LIN {X 0,Y 592.162,Z 615.177,A -85,B 0,C 180,E1 27814.744,E2 27814.744} C_VEL
LIN {X 0,Y 592.28,Z 584.282,A -85,B 0,C 180,E1 27811.546,E2 27811.546} C_VEL
LIN {X 0,Y 592.445,Z 553.985,A -85,B 0,C 180,E1 27808.355,E2 27808.355} C_VEL
LIN {X 0,Y 592.619,Z 523.409,A -85,B 0,C 180,E1 27805.063,E2 27805.063} C_VEL
LIN {X 0,Y 592.573,Z 507.534,A -85,B 0,C 180,E1 27803.314,E2 27803.314} C_VEL
LIN {X 0,Y 591.975,Z 505.143,A -85,B 0,C 180,E1 27802.966,E2 27802.966} C_VEL
LIN {X 0,Y 591.982,Z 505.056,A -85,B 0,C 180,E1 27800.079,E2 27800.079} C_VEL
LIN {X 0,Y 591.962,Z 505.055,A -85,B 0,C 180,E1 27796.819,E2 27796.819} C_VEL
LIN {X 0,Y 591.972,Z 505.055,A -85,B 0,C 180,E1 27793.959,E2 27793.959} C_VEL
LIN {X 0,Y 591.962,Z 505.055,A -85,B 0,C 180,E1 27790.668,E2 27790.668} C_VEL
LIN {X 0,Y 591.962,Z 505.055,A -85,B 0,C 180,E1 27787.874,E2 27787.874} C_VEL
LIN {X 0,Y 591.959,Z 505.055,A -85,B 0,C 180,E1 27784.488,E2 27784.488} C_VEL
LIN {X 0,Y 591.959,Z 505.055,A -85,B 0,C 180,E1 27781.666,E2 27781.666} C_VEL
LIN {X 0,Y 591.957,Z 505.053,A -85,B 0,C 180,E1 27778.313,E2 27778.313} C_VEL
LIN {X 0,Y 591.957,Z 505.055,A -85,B 0,C 180,E1 27775.515,E2 27775.515} C_VEL
LIN {X 0,Y 591.966,Z 505.054,A -85,B 0,C 180,E1 27772.187,E2 27772.187} C_VEL
LIN {X 0,Y 591.954,Z 505.055,A -85,B 0,C 180,E1 27769.439,E2 27769.439} C_VEL
LIN {X 0,Y 592,Z 505.054,A -85,B 0,C 180,E1 27766.292,E2 27766.292} C_VEL
LIN {X 0,Y 591.952,Z 505.055,A -85,B 0,C 180,E1 27763.426,E2 27763.426} C_VEL
LIN {X 0,Y 592.032,Z 505.053,A -85,B 0,C 180,E1 27760.304,E2 27760.304} C_VEL
LIN {X 0,Y 591.955,Z 505.054,A -85,B 0,C 180,E1 27757.297,E2 27757.297} C_VEL
LIN {X 0,Y 592.039,Z 505.051,A -85,B 0,C 180,E1 27754.159,E2 27754.159} C_VEL
LIN {X 0,Y 591.959,Z 505.054,A -85,B 0,C 180,E1 27751.096,E2 27751.096} C_VEL
LIN {X 0,Y 592.041,Z 505.051,A -85,B 0,C 180,E1 27748.002,E2 27748.002} C_VEL
LIN {X 0,Y 591.961,Z 505.052,A -85,B 0,C 180,E1 27744.91,E2 27744.91} C_VEL
LIN {X 0,Y 592.039,Z 505.053,A -85,B 0,C 180,E1 27741.811,E2 27741.811} C_VEL
LIN {X 0,Y 591.965,Z 505.051,A -85,B 0,C 180,E1 27738.719,E2 27738.719} C_VEL
LIN {X 0,Y 592.039,Z 505.051,A -85,B 0,C 180,E1 27735.577,E2 27735.577} C_VEL
LIN {X 0,Y 591.968,Z 505.053,A -85,B 0,C 180,E1 27732.486,E2 27732.486} C_VEL
LIN {X 0,Y 592.034,Z 505.048,A -85,B 0,C 180,E1 27729.331,E2 27729.331} C_VEL
LIN {X 0,Y 591.971,Z 505.052,A -85,B 0,C 180,E1 27726.303,E2 27726.303} C_VEL
LIN {X 0,Y 592.038,Z 505.05,A -85,B 0,C 180,E1 27723.195,E2 27723.195} C_VEL
LIN {X 0,Y 591.974,Z 505.049,A -85,B 0,C 180,E1 27720.097,E2 27720.097} C_VEL
LIN {X 0,Y 592.033,Z 505.05,A -85,B 0,C 180,E1 27716.902,E2 27716.902} C_VEL
LIN {X 0,Y 591.979,Z 505.052,A -85,B 0,C 180,E1 27713.795,E2 27713.795} C_VEL
LIN {X 0,Y 592.024,Z 505.048,A -85,B 0,C 180,E1 27710.571,E2 27710.571} C_VEL
LIN {X 0,Y 591.986,Z 505.053,A -85,B 0,C 180,E1 27707.515,E2 27707.515} C_VEL
LIN {X 0,Y 592.009,Z 505.048,A -85,B 0,C 180,E1 27704.222,E2 27704.222} C_VEL
LIN {X 0,Y 591.997,Z 505.054,A -85,B 0,C 180,E1 27701.18,E2 27701.18} C_VEL
LIN {X 0,Y 591.997,Z 505.049,A -85,B 0,C 180,E1 27697.875,E2 27697.875} C_VEL
LIN {X 0,Y 592.016,Z 505.054,A -85,B 0,C 180,E1 27694.811,E2 27694.811} C_VEL
LIN {X 0,Y 591.991,Z 505.05,A -85,B 0,C 180,E1 27691.557,E2 27691.557} C_VEL
LIN {X 0,Y 592.028,Z 505.055,A -85,B 0,C 180,E1 27688.52,E2 27688.52} C_VEL
LIN {X 0,Y 591.99,Z 505.049,A -85,B 0,C 180,E1 27685.307,E2 27685.307} C_VEL
LIN {X 0,Y 592.038,Z 505.053,A -85,B 0,C 180,E1 27682.19,E2 27682.19} C_VEL
LIN {X 0,Y 591.992,Z 505.05,A -85,B 0,C 180,E1 27679.019,E2 27679.019} C_VEL
LIN {X 0,Y 592.035,Z 505.051,A -85,B 0,C 180,E1 27675.866,E2 27675.866} C_VEL
LIN {X 0,Y 591.992,Z 505.051,A -85,B 0,C 180,E1 27672.718,E2 27672.718} C_VEL
LIN {X 0,Y 592.035,Z 505.051,A -85,B 0,C 180,E1 27669.636,E2 27669.636} C_VEL
LIN {X 0,Y 591.995,Z 505.051,A -85,B 0,C 180,E1 27666.476,E2 27666.476} C_VEL
LIN {X 0,Y 592.035,Z 505.046,A -85,B 0,C 180,E1 27663.282,E2 27663.282} C_VEL
LIN {X 0,Y 592.026,Z 505.235,A -85,B 0,C 180,E1 27660.534,E2 27660.534} C_VEL
LIN {X 0,Y 593.397,Z 509.911,A -85,B 0,C 180,E1 27660.083,E2 27660.083} C_VEL
LIN {X 0,Y 593.093,Z 554.015,A -85,B 0,C 180,E1 27657.021,E2 27657.021} C_VEL
LIN {X 0,Y 592.85,Z 599.79,A -85,B 0,C 180,E1 27653.922,E2 27653.922} C_VEL
LIN {X 0,Y 592.854,Z 615.059,A -85,B 0,C 180,E1 27652.928,E2 27652.928} C_VEL
LIN {X 0,Y 593.106,Z 625.3,A -85,B 0,C 180,E1 27652.782,E2 27652.782} C_VEL
LIN {X 0,Y 592.846,Z 824.35,A -85,B 0,C 180,E1 27650.226,E2 27650.226} C_VEL
LIN {X 0,Y 592.749,Z 843.327,A -85,B 0,C 180,E1 27649.797,E2 27649.797} C_VEL
LIN {X 0,Y 592.671,Z 861.42,A -85,B 0,C 180,E1 27649.206,E2 27649.206} C_VEL
LIN {X 0,Y 592.541,Z 879.065,A -85,B 0,C 180,E1 27648.444,E2 27648.444} C_VEL
LIN {X 0,Y 592.459,Z 895.697,A -85,B 0,C 180,E1 27647.538,E2 27647.538} C_VEL
LIN {X 0,Y 592.342,Z 911.642,A -85,B 0,C 180,E1 27646.474,E2 27646.474} C_VEL
LIN {X 0,Y 592.23,Z 926.565,A -85,B 0,C 180,E1 27645.27,E2 27645.27} C_VEL
LIN {X 0,Y 592.131,Z 940.02,A -85,B 0,C 180,E1 27643.973,E2 27643.973} C_VEL
LIN {X 0,Y 592.058,Z 952.908,A -85,B 0,C 180,E1 27642.484,E2 27642.484} C_VEL
LIN {X 0,Y 591.999,Z 964.225,A -85,B 0,C 180,E1 27640.904,E2 27640.904} C_VEL
LIN {X 0,Y 591.954,Z 973.989,A -85,B 0,C 180,E1 27639.234,E2 27639.234} C_VEL
LIN {X 0,Y 591.935,Z 981.771,A -85,B 0,C 180,E1 27637.571,E2 27637.571} C_VEL
LIN {X 0,Y 591.913,Z 988.263,A -85,B 0,C 180,E1 27635.767,E2 27635.767} C_VEL
LIN {X 0,Y 591.918,Z 992.872,A -85,B 0,C 180,E1 27633.972,E2 27633.972} C_VEL
LIN {X 0,Y 591.917,Z 995.787,A -85,B 0,C 180,E1 27632.131,E2 27632.131} C_VEL
LIN {X 0,Y 591.908,Z 996.939,A -85,B 0,C 180,E1 27630.292,E2 27630.292} C_VEL
LIN {X 0,Y 591.915,Z 996.349,A -85,B 0,C 180,E1 27628.453,E2 27628.453} C_VEL
LIN {X 0,Y 591.907,Z 994.008,A -85,B 0,C 180,E1 27626.612,E2 27626.612} C_VEL
LIN {X 0,Y 591.912,Z 990.101,A -85,B 0,C 180,E1 27624.865,E2 27624.865} C_VEL
LIN {X 0,Y 591.928,Z 984.474,A -85,B 0,C 180,E1 27623.114,E2 27623.114} C_VEL
LIN {X 0,Y 591.941,Z 977.432,A -85,B 0,C 180,E1 27621.454,E2 27621.454} C_VEL
LIN {X 0,Y 591.976,Z 968.523,A -85,B 0,C 180,E1 27619.787,E2 27619.787} C_VEL
LIN {X 0,Y 592.024,Z 958.162,A -85,B 0,C 180,E1 27618.211,E2 27618.211} C_VEL
LIN {X 0,Y 592.093,Z 946.367,A -85,B 0,C 180,E1 27616.725,E2 27616.725} C_VEL
LIN {X 0,Y 592.193,Z 932.605,A -85,B 0,C 180,E1 27615.282,E2 27615.282} C_VEL
LIN {X 0,Y 592.305,Z 917.629,A -85,B 0,C 180,E1 27613.981,E2 27613.981} C_VEL
LIN {X 0,Y 592.421,Z 901.463,A -85,B 0,C 180,E1 27612.824,E2 27612.824} C_VEL
LIN {X 0,Y 592.508,Z 885.089,A -85,B 0,C 180,E1 27611.863,E2 27611.863} C_VEL
LIN {X 0,Y 592.648,Z 868.165,A -85,B 0,C 180,E1 27611.063,E2 27611.063} C_VEL
LIN {X 0,Y 592.725,Z 849.831,A -85,B 0,C 180,E1 27610.395,E2 27610.395} C_VEL
LIN {X 0,Y 592.818,Z 831.296,A -85,B 0,C 180,E1 27609.91,E2 27609.91} C_VEL
LIN {X 0,Y 592.884,Z 811.474,A -85,B 0,C 180,E1 27609.586,E2 27609.586} C_VEL
LIN {X 0,Y 592.949,Z 615.757,A -85,B 0,C 180,E1 27607.089,E2 27607.089} C_VEL
LIN {X 0,Y 592.795,Z 613.121,A -85,B 0,C 180,E1 27606.967,E2 27606.967} C_VEL
LIN {X 0,Y 593.04,Z 564.292,A -85,B 0,C 180,E1 27603.682,E2 27603.682} C_VEL
LIN {X 0,Y 593.332,Z 519.662,A -85,B 0,C 180,E1 27600.602,E2 27600.602} C_VEL
LIN {X 0,Y 593.226,Z 508.987,A -85,B 0,C 180,E1 27599.842,E2 27599.842} C_VEL
LIN {X 0,Y 592.027,Z 505.245,A -85,B 0,C 180,E1 27599.466,E2 27599.466} C_VEL
LIN {X 0,Y 592.034,Z 505.055,A -85,B 0,C 180,E1 27596.367,E2 27596.367} C_VEL
LIN {X 0,Y 592.003,Z 505.05,A -85,B 0,C 180,E1 27593.166,E2 27593.166} C_VEL
LIN {X 0,Y 592.006,Z 505.053,A -85,B 0,C 180,E1 27589.827,E2 27589.827} C_VEL
LIN {X 0,Y 592.021,Z 505.048,A -85,B 0,C 180,E1 27586.712,E2 27586.712} C_VEL
LIN {X 0,Y 591.992,Z 505.054,A -85,B 0,C 180,E1 27583.559,E2 27583.559} C_VEL
LIN {X 0,Y 592.034,Z 505.048,A -85,B 0,C 180,E1 27580.396,E2 27580.396} C_VEL
LIN {X 0,Y 591.978,Z 505.053,A -85,B 0,C 180,E1 27577.205,E2 27577.205} C_VEL
LIN {X 0,Y 592.04,Z 505.05,A -85,B 0,C 180,E1 27574.104,E2 27574.104} C_VEL
LIN {X 0,Y 591.971,Z 505.053,A -85,B 0,C 180,E1 27571.008,E2 27571.008} C_VEL
LIN {X 0,Y 592.033,Z 505.051,A -85,B 0,C 180,E1 27567.972,E2 27567.972} C_VEL
LIN {X 0,Y 591.964,Z 505.053,A -85,B 0,C 180,E1 27564.871,E2 27564.871} C_VEL
LIN {X 0,Y 592.012,Z 505.052,A -85,B 0,C 180,E1 27561.916,E2 27561.916} C_VEL
LIN {X 0,Y 591.958,Z 505.054,A -85,B 0,C 180,E1 27558.719,E2 27558.719} C_VEL
LIN {X 0,Y 592.007,Z 505.054,A -85,B 0,C 180,E1 27555.722,E2 27555.722} C_VEL
LIN {X 0,Y 591.95,Z 505.055,A -85,B 0,C 180,E1 27552.585,E2 27552.585} C_VEL
LIN {X 0,Y 591.981,Z 505.055,A -85,B 0,C 180,E1 27549.724,E2 27549.724} C_VEL
LIN {X 0,Y 591.956,Z 505.055,A -85,B 0,C 180,E1 27546.498,E2 27546.498} C_VEL
LIN {X 0,Y 591.977,Z 505.054,A -85,B 0,C 180,E1 27543.68,E2 27543.68} C_VEL
LIN {X 0,Y 591.967,Z 505.052,A -85,B 0,C 180,E1 27540.387,E2 27540.387} C_VEL
LIN {X 0,Y 591.978,Z 505.055,A -85,B 0,C 180,E1 27537.58,E2 27537.58} C_VEL
LIN {X 0,Y 591.977,Z 505.052,A -85,B 0,C 180,E1 27534.281,E2 27534.281} C_VEL
LIN {X 0,Y 591.99,Z 505.054,A -85,B 0,C 180,E1 27531.354,E2 27531.354} C_VEL
LIN {X 0,Y 591.974,Z 505.051,A -85,B 0,C 180,E1 27530.026,E2 27530.026} C_VEL
LIN {X 0,Y 590.981,Z 505.18,A -85,B 0,C 180,E1 27529.281,E2 27529.281} C_VEL
LIN {X 0,Y 584.627,Z 505.979,A -85,B 0,C 180,E1 27527.188,E2 27527.188} C_VEL
LIN {X 0,Y 584.1,Z 506.039,A -85,B 0,C 180,E1 27526.644,E2 27526.644} C_VEL
LIN {X 0,Y 584.04,Z 506.042,A -85,B 0,C 180,E1 27523.489,E2 27523.489} C_VEL
LIN {X 0,Y 584.089,Z 506.038,A -85,B 0,C 180,E1 27520.288,E2 27520.288} C_VEL
LIN {X 0,Y 584.049,Z 506.042,A -85,B 0,C 180,E1 27517.238,E2 27517.238} C_VEL
LIN {X 0,Y 584.082,Z 506.037,A -85,B 0,C 180,E1 27513.977,E2 27513.977} C_VEL
LIN {X 0,Y 584.074,Z 506.044,A -85,B 0,C 180,E1 27510.798,E2 27510.798} C_VEL
LIN {X 0,Y 584.062,Z 506.039,A -85,B 0,C 180,E1 27507.483,E2 27507.483} C_VEL
LIN {X 0,Y 584.098,Z 506.043,A -85,B 0,C 180,E1 27504.287,E2 27504.287} C_VEL
LIN {X 0,Y 584.061,Z 506.041,A -85,B 0,C 180,E1 27501.077,E2 27501.077} C_VEL
LIN {X 0,Y 584.092,Z 506.04,A -85,B 0,C 180,E1 27497.974,E2 27497.974} C_VEL
LIN {X 0,Y 584.11,Z 506.324,A -85,B 0,C 180,E1 27497.17,E2 27497.17} C_VEL
LIN {X 0,Y 585.103,Z 511.061,A -85,B 0,C 180,E1 27496.567,E2 27496.567} C_VEL
LIN {X 0,Y 584.831,Z 540.901,A -85,B 0,C 180,E1 27493.274,E2 27493.274} C_VEL
LIN {X 0,Y 584.591,Z 571.112,A -85,B 0,C 180,E1 27490.017,E2 27490.017} C_VEL
LIN {X 0,Y 584.393,Z 601.721,A -85,B 0,C 180,E1 27486.781,E2 27486.781} C_VEL
LIN {X 0,Y 584.226,Z 632.278,A -85,B 0,C 180,E1 27483.613,E2 27483.613} C_VEL
LIN {X 0,Y 584.414,Z 634.271,A -85,B 0,C 180,E1 27483.528,E2 27483.528} C_VEL
LIN {X 0,Y 584.38,Z 744.506,A -85,B 0,C 180,E1 27482.14,E2 27482.14} C_VEL
LIN {X 0,Y 584.362,Z 759.323,A -85,B 0,C 180,E1 27481.771,E2 27481.771} C_VEL
LIN {X 0,Y 584.292,Z 773.461,A -85,B 0,C 180,E1 27481.227,E2 27481.227} C_VEL
LIN {X 0,Y 584.186,Z 786.407,A -85,B 0,C 180,E1 27480.548,E2 27480.548} C_VEL
LIN {X 0,Y 584.122,Z 799.494,A -85,B 0,C 180,E1 27479.645,E2 27479.645} C_VEL
LIN {X 0,Y 584.051,Z 810.723,A -85,B 0,C 180,E1 27478.638,E2 27478.638} C_VEL
LIN {X 0,Y 583.999,Z 820.156,A -85,B 0,C 180,E1 27477.585,E2 27477.585} C_VEL
LIN {X 0,Y 583.959,Z 829.004,A -85,B 0,C 180,E1 27476.321,E2 27476.321} C_VEL
LIN {X 0,Y 583.932,Z 836.418,A -85,B 0,C 180,E1 27474.908,E2 27474.908} C_VEL
LIN {X 0,Y 583.921,Z 841.635,A -85,B 0,C 180,E1 27473.51,E2 27473.51} C_VEL
LIN {X 0,Y 583.919,Z 845.039,A -85,B 0,C 180,E1 27472.123,E2 27472.123} C_VEL
LIN {X 0,Y 583.918,Z 846.85,A -85,B 0,C 180,E1 27470.547,E2 27470.547} C_VEL
LIN {X 0,Y 583.915,Z 846.641,A -85,B 0,C 180,E1 27469.053,E2 27469.053} C_VEL
LIN {X 0,Y 583.916,Z 844.748,A -85,B 0,C 180,E1 27467.64,E2 27467.64} C_VEL
LIN {X 0,Y 583.922,Z 840.813,A -85,B 0,C 180,E1 27466.134,E2 27466.134} C_VEL
LIN {X 0,Y 583.936,Z 834.904,A -85,B 0,C 180,E1 27464.677,E2 27464.677} C_VEL
LIN {X 0,Y 583.957,Z 827.562,A -85,B 0,C 180,E1 27463.362,E2 27463.362} C_VEL
LIN {X 0,Y 584.01,Z 818.777,A -85,B 0,C 180,E1 27462.152,E2 27462.152} C_VEL
LIN {X 0,Y 584.077,Z 807.494,A -85,B 0,C 180,E1 27460.952,E2 27460.952} C_VEL
LIN {X 0,Y 584.146,Z 795.357,A -85,B 0,C 180,E1 27459.953,E2 27459.953} C_VEL
LIN {X 0,Y 584.223,Z 782.843,A -85,B 0,C 180,E1 27459.156,E2 27459.156} C_VEL
LIN {X 0,Y 584.317,Z 769.527,A -85,B 0,C 180,E1 27458.51,E2 27458.51} C_VEL
LIN {X 0,Y 584.389,Z 754.072,A -85,B 0,C 180,E1 27457.986,E2 27457.986} C_VEL
LIN {X 0,Y 584.423,Z 738.839,A -85,B 0,C 180,E1 27457.678,E2 27457.678} C_VEL
LIN {X 0,Y 584.324,Z 633.555,A -85,B 0,C 180,E1 27456.369,E2 27456.369} C_VEL
LIN {X 0,Y 584.237,Z 631.108,A -85,B 0,C 180,E1 27456.188,E2 27456.188} C_VEL
LIN {X 0,Y 584.376,Z 599.932,A -85,B 0,C 180,E1 27452.941,E2 27452.941} C_VEL
LIN {X 0,Y 584.614,Z 569.348,A -85,B 0,C 180,E1 27449.705,E2 27449.705} C_VEL
LIN {X 0,Y 584.838,Z 539.388,A -85,B 0,C 180,E1 27446.471,E2 27446.471} C_VEL
LIN {X 0,Y 585.105,Z 510.476,A -85,B 0,C 180,E1 27443.277,E2 27443.277} C_VEL
LIN {X 0,Y 584.036,Z 506.181,A -85,B 0,C 180,E1 27442.697,E2 27442.697} C_VEL
LIN {X 0,Y 584.094,Z 506.043,A -85,B 0,C 180,E1 27439.645,E2 27439.645} C_VEL
LIN {X 0,Y 584.015,Z 506.044,A -85,B 0,C 180,E1 27436.519,E2 27436.519} C_VEL
LIN {X 0,Y 584.094,Z 506.045,A -85,B 0,C 180,E1 27433.389,E2 27433.389} C_VEL
LIN {X 0,Y 584.012,Z 506.043,A -85,B 0,C 180,E1 27430.29,E2 27430.29} C_VEL
LIN {X 0,Y 584.088,Z 506.041,A -85,B 0,C 180,E1 27427.241,E2 27427.241} C_VEL
LIN {X 0,Y 584.008,Z 506.044,A -85,B 0,C 180,E1 27424.115,E2 27424.115} C_VEL
LIN {X 0,Y 584.085,Z 506.041,A -85,B 0,C 180,E1 27421.016,E2 27421.016} C_VEL
LIN {X 0,Y 584.006,Z 506.041,A -85,B 0,C 180,E1 27417.939,E2 27417.939} C_VEL
LIN {X 0,Y 584.085,Z 506.046,A -85,B 0,C 180,E1 27414.89,E2 27414.89} C_VEL
LIN {X 0,Y 584.01,Z 506.043,A -85,B 0,C 180,E1 27411.798,E2 27411.798} C_VEL
LIN {X 0,Y 584.093,Z 506.044,A -85,B 0,C 180,E1 27408.72,E2 27408.72} C_VEL
LIN {X 0,Y 584.015,Z 506.043,A -85,B 0,C 180,E1 27405.695,E2 27405.695} C_VEL
LIN {X 0,Y 584.063,Z 506.044,A -85,B 0,C 180,E1 27402.747,E2 27402.747} C_VEL
LIN {X 0,Y 584.019,Z 506.042,A -85,B 0,C 180,E1 27399.56,E2 27399.56} C_VEL
LIN {X 0,Y 584.066,Z 506.044,A -85,B 0,C 180,E1 27396.566,E2 27396.566} C_VEL
LIN {X 0,Y 584.026,Z 506.04,A -85,B 0,C 180,E1 27393.454,E2 27393.454} C_VEL
LIN {X 0,Y 584.048,Z 506.043,A -85,B 0,C 180,E1 27390.561,E2 27390.561} C_VEL
LIN {X 0,Y 584.032,Z 506.039,A -85,B 0,C 180,E1 27387.311,E2 27387.311} C_VEL
LIN {X 0,Y 584.051,Z 506.041,A -85,B 0,C 180,E1 27384.367,E2 27384.367} C_VEL
LIN {X 0,Y 584.031,Z 506.041,A -85,B 0,C 180,E1 27381.071,E2 27381.071} C_VEL
LIN {X 0,Y 584.068,Z 506.041,A -85,B 0,C 180,E1 27378.051,E2 27378.051} C_VEL
LIN {X 0,Y 584.034,Z 506.041,A -85,B 0,C 180,E1 27374.88,E2 27374.88} C_VEL
LIN {X 0,Y 584.072,Z 506.044,A -85,B 0,C 180,E1 27371.855,E2 27371.855} C_VEL
LIN {X 0,Y 584.036,Z 506.036,A -85,B 0,C 180,E1 27368.665,E2 27368.665} C_VEL
LIN {X 0,Y 584.068,Z 506.043,A -85,B 0,C 180,E1 27365.698,E2 27365.698} C_VEL
LIN {X 0,Y 584.038,Z 506.039,A -85,B 0,C 180,E1 27362.453,E2 27362.453} C_VEL
LIN {X 0,Y 584.082,Z 506.04,A -85,B 0,C 180,E1 27359.412,E2 27359.412} C_VEL
LIN {X 0,Y 584.038,Z 506.041,A -85,B 0,C 180,E1 27356.172,E2 27356.172} C_VEL
LIN {X 0,Y 584.101,Z 506.038,A -85,B 0,C 180,E1 27353.019,E2 27353.019} C_VEL
LIN {X 0,Y 584.039,Z 506.04,A -85,B 0,C 180,E1 27349.84,E2 27349.84} C_VEL
LIN {X 0,Y 584.1,Z 506.038,A -85,B 0,C 180,E1 27346.74,E2 27346.74} C_VEL
LIN {X 0,Y 584.042,Z 506.04,A -85,B 0,C 180,E1 27343.592,E2 27343.592} C_VEL
LIN {X 0,Y 584.098,Z 506.036,A -85,B 0,C 180,E1 27340.396,E2 27340.396} C_VEL
LIN {X 0,Y 584.049,Z 506.041,A -85,B 0,C 180,E1 27337.238,E2 27337.238} C_VEL
LIN {X 0,Y 584.082,Z 506.035,A -85,B 0,C 180,E1 27333.983,E2 27333.983} C_VEL
LIN {X 0,Y 584.068,Z 506.043,A -85,B 0,C 180,E1 27330.798,E2 27330.798} C_VEL
LIN {X 0,Y 584.058,Z 506.038,A -85,B 0,C 180,E1 27327.484,E2 27327.484} C_VEL
LIN {X 0,Y 584.1,Z 506.042,A -85,B 0,C 180,E1 27324.287,E2 27324.287} C_VEL
LIN {X 0,Y 584.052,Z 506.038,A -85,B 0,C 180,E1 27321.077,E2 27321.077} C_VEL
LIN {X 0,Y 584.098,Z 506.041,A -85,B 0,C 180,E1 27317.977,E2 27317.977} C_VEL
LIN {X 0,Y 584.054,Z 506.038,A -85,B 0,C 180,E1 27314.852,E2 27314.852} C_VEL
LIN {X 0,Y 584.096,Z 506.041,A -85,B 0,C 180,E1 27311.725,E2 27311.725} C_VEL
LIN {X 0,Y 584.056,Z 506.041,A -85,B 0,C 180,E1 27308.524,E2 27308.524} C_VEL
LIN {X 0,Y 584.096,Z 506.037,A -85,B 0,C 180,E1 27305.261,E2 27305.261} C_VEL
LIN {X 0,Y 584.067,Z 506.039,A -85,B 0,C 180,E1 27302.05,E2 27302.05} C_VEL
LIN {X 0,Y 584.131,Z 506.345,A -85,B 0,C 180,E1 27300.896,E2 27300.896} C_VEL
LIN {X 0,Y 586.143,Z 513.061,A -85,B 0,C 180,E1 27300.268,E2 27300.268} C_VEL
LIN {X 0,Y 585.694,Z 557.086,A -85,B 0,C 180,E1 27297.176,E2 27297.176} C_VEL
LIN {X 0,Y 585.33,Z 602.057,A -85,B 0,C 180,E1 27294.095,E2 27294.095} C_VEL
LIN {X 0,Y 585.344,Z 615.25,A -85,B 0,C 180,E1 27293.236,E2 27293.236} C_VEL
LIN {X 0,Y 585.737,Z 621.221,A -85,B 0,C 180,E1 27293.138,E2 27293.138} C_VEL
LIN {X 0,Y 585.336,Z 824.35,A -85,B 0,C 180,E1 27290.498,E2 27290.498} C_VEL
LIN {X 0,Y 585.201,Z 843.326,A -85,B 0,C 180,E1 27290.064,E2 27290.064} C_VEL
LIN {X 0,Y 585.074,Z 861.418,A -85,B 0,C 180,E1 27289.465,E2 27289.465} C_VEL
LIN {X 0,Y 584.891,Z 879.061,A -85,B 0,C 180,E1 27288.694,E2 27288.694} C_VEL
LIN {X 0,Y 584.738,Z 896.222,A -85,B 0,C 180,E1 27287.744,E2 27287.744} C_VEL
LIN {X 0,Y 584.561,Z 912.241,A -85,B 0,C 180,E1 27286.653,E2 27286.653} C_VEL
LIN {X 0,Y 584.393,Z 927.097,A -85,B 0,C 180,E1 27285.431,E2 27285.431} C_VEL
LIN {X 0,Y 584.241,Z 940.946,A -85,B 0,C 180,E1 27284.065,E2 27284.065} C_VEL
LIN {X 0,Y 584.129,Z 953.684,A -85,B 0,C 180,E1 27282.556,E2 27282.556} C_VEL
LIN {X 0,Y 584.041,Z 964.864,A -85,B 0,C 180,E1 27280.955,E2 27280.955} C_VEL
LIN {X 0,Y 583.976,Z 974.507,A -85,B 0,C 180,E1 27279.262,E2 27279.262} C_VEL
LIN {X 0,Y 583.942,Z 982.403,A -85,B 0,C 180,E1 27277.521,E2 27277.521} C_VEL
LIN {X 0,Y 583.918,Z 988.409,A -85,B 0,C 180,E1 27275.799,E2 27275.799} C_VEL
LIN {X 0,Y 583.919,Z 992.873,A -85,B 0,C 180,E1 27274.027,E2 27274.027} C_VEL
LIN {X 0,Y 583.916,Z 995.788,A -85,B 0,C 180,E1 27272.16,E2 27272.16} C_VEL
LIN {X 0,Y 583.907,Z 996.939,A -85,B 0,C 180,E1 27270.296,E2 27270.296} C_VEL
LIN {X 0,Y 583.915,Z 996.35,A -85,B 0,C 180,E1 27268.431,E2 27268.431} C_VEL
LIN {X 0,Y 583.907,Z 994.008,A -85,B 0,C 180,E1 27266.566,E2 27266.566} C_VEL
LIN {X 0,Y 583.916,Z 990.102,A -85,B 0,C 180,E1 27264.795,E2 27264.795} C_VEL
LIN {X 0,Y 583.934,Z 984.474,A -85,B 0,C 180,E1 27263.019,E2 27263.019} C_VEL
LIN {X 0,Y 583.956,Z 977.433,A -85,B 0,C 180,E1 27261.336,E2 27261.336} C_VEL
LIN {X 0,Y 584.015,Z 968.524,A -85,B 0,C 180,E1 27259.646,E2 27259.646} C_VEL
LIN {X 0,Y 584.086,Z 958.163,A -85,B 0,C 180,E1 27258.048,E2 27258.048} C_VEL
LIN {X 0,Y 584.195,Z 946.367,A -85,B 0,C 180,E1 27256.542,E2 27256.542} C_VEL
LIN {X 0,Y 584.342,Z 932.604,A -85,B 0,C 180,E1 27255.08,E2 27255.08} C_VEL
LIN {X 0,Y 584.507,Z 917.631,A -85,B 0,C 180,E1 27253.761,E2 27253.761} C_VEL
LIN {X 0,Y 584.685,Z 901.465,A -85,B 0,C 180,E1 27252.589,E2 27252.589} C_VEL
LIN {X 0,Y 584.833,Z 884.708,A -85,B 0,C 180,E1 27251.596,E2 27251.596} C_VEL
LIN {X 0,Y 585.033,Z 867.87,A -85,B 0,C 180,E1 27250.795,E2 27250.795} C_VEL
LIN {X 0,Y 585.161,Z 849.726,A -85,B 0,C 180,E1 27250.128,E2 27250.128} C_VEL
LIN {X 0,Y 585.295,Z 831.296,A -85,B 0,C 180,E1 27249.641,E2 27249.641} C_VEL
LIN {X 0,Y 585.385,Z 811.421,A -85,B 0,C 180,E1 27249.312,E2 27249.312} C_VEL
LIN {X 0,Y 585.577,Z 616.821,A -85,B 0,C 180,E1 27246.798,E2 27246.798} C_VEL
LIN {X 0,Y 585.259,Z 613.94,A -85,B 0,C 180,E1 27246.707,E2 27246.707} C_VEL
LIN {X 0,Y 585.628,Z 565.867,A -85,B 0,C 180,E1 27243.432,E2 27243.432} C_VEL
LIN {X 0,Y 586.068,Z 520.64,A -85,B 0,C 180,E1 27240.271,E2 27240.271} C_VEL
LIN {X 0,Y 585.909,Z 511.612,A -85,B 0,C 180,E1 27239.614,E2 27239.614} C_VEL
LIN {X 0,Y 584.135,Z 506.368,A -85,B 0,C 180,E1 27239.107,E2 27239.107} C_VEL
LIN {X 0,Y 584.086,Z 506.042,A -85,B 0,C 180,E1 27238.185,E2 27238.185} C_VEL
LIN {X 0,Y 584.092,Z 506.038,A -85,B 0,C 180,E1 27234.893,E2 27234.893} C_VEL
LIN {X 0,Y 584.055,Z 506.042,A -85,B 0,C 180,E1 27231.634,E2 27231.634} C_VEL
LIN {X 0,Y 584.101,Z 506.037,A -85,B 0,C 180,E1 27228.518,E2 27228.518} C_VEL
LIN {X 0,Y 584.047,Z 506.042,A -85,B 0,C 180,E1 27225.412,E2 27225.412} C_VEL
LIN {X 0,Y 584.098,Z 506.04,A -85,B 0,C 180,E1 27222.279,E2 27222.279} C_VEL
LIN {X 0,Y 584.039,Z 506.04,A -85,B 0,C 180,E1 27219.156,E2 27219.156} C_VEL
LIN {X 0,Y 584.102,Z 506.041,A -85,B 0,C 180,E1 27216.076,E2 27216.076} C_VEL
LIN {X 0,Y 584.034,Z 506.041,A -85,B 0,C 180,E1 27212.984,E2 27212.984} C_VEL
LIN {X 0,Y 584.101,Z 506.044,A -85,B 0,C 180,E1 27209.763,E2 27209.763} C_VEL
LIN {X 0,Y 584.027,Z 506.042,A -85,B 0,C 180,E1 27206.65,E2 27206.65} C_VEL
LIN {X 0,Y 584.083,Z 506.044,A -85,B 0,C 180,E1 27203.507,E2 27203.507} C_VEL
LIN {X 0,Y 584.019,Z 506.043,A -85,B 0,C 180,E1 27200.546,E2 27200.546} C_VEL
LIN {X 0,Y 584.088,Z 506.045,A -85,B 0,C 180,E1 27197.432,E2 27197.432} C_VEL
LIN {X 0,Y 584.011,Z 506.041,A -85,B 0,C 180,E1 27194.374,E2 27194.374} C_VEL
LIN {X 0,Y 584.079,Z 506.043,A -85,B 0,C 180,E1 27191.25,E2 27191.25} C_VEL
LIN {X 0,Y 584.011,Z 506.044,A -85,B 0,C 180,E1 27188.169,E2 27188.169} C_VEL
LIN {X 0,Y 584.074,Z 506.041,A -85,B 0,C 180,E1 27185.008,E2 27185.008} C_VEL
LIN {X 0,Y 584.02,Z 506.044,A -85,B 0,C 180,E1 27181.962,E2 27181.962} C_VEL
LIN {X 0,Y 584.079,Z 506.041,A -85,B 0,C 180,E1 27178.823,E2 27178.823} C_VEL
LIN {X 0,Y 584.028,Z 506.042,A -85,B 0,C 180,E1 27175.778,E2 27175.778} C_VEL
LIN {X 0,Y 584.069,Z 506.04,A -85,B 0,C 180,E1 27172.524,E2 27172.524} C_VEL
LIN {X 0,Y 584.037,Z 506.041,A -85,B 0,C 180,E1 27169.544,E2 27169.544} C_VEL
LIN {X 0,Y 584.1,Z 506.039,A -85,B 0,C 180,E1 27166.644,E2 27166.644} C_VEL
LIN {X 0,Y 583.094,Z 506.161,A -85,B 0,C 180,E1 27165.889,E2 27165.889} C_VEL
LIN {X 0,Y 576.624,Z 506.966,A -85,B 0,C 180,E1 27163.768,E2 27163.768} C_VEL
LIN {X 0,Y 576.116,Z 507.032,A -85,B 0,C 180,E1 27163.216,E2 27163.216} C_VEL
LIN {X 0,Y 576.114,Z 507.028,A -85,B 0,C 180,E1 27159.853,E2 27159.853} C_VEL
LIN {X 0,Y 576.158,Z 507.033,A -85,B 0,C 180,E1 27156.692,E2 27156.692} C_VEL
LIN {X 0,Y 576.113,Z 507.029,A -85,B 0,C 180,E1 27153.51,E2 27153.51} C_VEL
LIN {X 0,Y 576.16,Z 507.031,A -85,B 0,C 180,E1 27150.357,E2 27150.357} C_VEL
LIN {X 0,Y 576.117,Z 507.03,A -85,B 0,C 180,E1 27147.129,E2 27147.129} C_VEL
LIN {X 0,Y 576.159,Z 507.028,A -85,B 0,C 180,E1 27143.959,E2 27143.959} C_VEL
LIN {X 0,Y 576.132,Z 507.033,A -85,B 0,C 180,E1 27140.695,E2 27140.695} C_VEL
LIN {X 0,Y 576.175,Z 507.205,A -85,B 0,C 180,E1 27137.513,E2 27137.513} C_VEL
LIN {X 0,Y 577.519,Z 513.123,A -85,B 0,C 180,E1 27136.717,E2 27136.717} C_VEL
LIN {X 0,Y 577.148,Z 542.307,A -85,B 0,C 180,E1 27133.447,E2 27133.447} C_VEL
LIN {X 0,Y 576.825,Z 572.035,A -85,B 0,C 180,E1 27130.199,E2 27130.199} C_VEL
LIN {X 0,Y 576.561,Z 602.613,A -85,B 0,C 180,E1 27126.921,E2 27126.921} C_VEL
LIN {X 0,Y 576.336,Z 632.336,A -85,B 0,C 180,E1 27123.798,E2 27123.798} C_VEL
LIN {X 0,Y 576.561,Z 634.544,A -85,B 0,C 180,E1 27123.713,E2 27123.713} C_VEL
LIN {X 0,Y 576.557,Z 744.44,A -85,B 0,C 180,E1 27122.31,E2 27122.31} C_VEL
LIN {X 0,Y 576.52,Z 759.434,A -85,B 0,C 180,E1 27121.931,E2 27121.931} C_VEL
LIN {X 0,Y 576.422,Z 774.132,A -85,B 0,C 180,E1 27121.353,E2 27121.353} C_VEL
LIN {X 0,Y 576.279,Z 787.636,A -85,B 0,C 180,E1 27120.618,E2 27120.618} C_VEL
LIN {X 0,Y 576.193,Z 799.845,A -85,B 0,C 180,E1 27119.751,E2 27119.751} C_VEL
LIN {X 0,Y 576.099,Z 811.011,A -85,B 0,C 180,E1 27118.73,E2 27118.73} C_VEL
LIN {X 0,Y 576.033,Z 819.947,A -85,B 0,C 180,E1 27117.718,E2 27117.718} C_VEL
LIN {X 0,Y 575.973,Z 828.496,A -85,B 0,C 180,E1 27116.492,E2 27116.492} C_VEL
LIN {X 0,Y 575.941,Z 835.541,A -85,B 0,C 180,E1 27115.168,E2 27115.168} C_VEL
LIN {X 0,Y 575.924,Z 841.065,A -85,B 0,C 180,E1 27113.748,E2 27113.748} C_VEL
LIN {X 0,Y 575.917,Z 844.884,A -85,B 0,C 180,E1 27112.236,E2 27112.236} C_VEL
LIN {X 0,Y 575.917,Z 846.728,A -85,B 0,C 180,E1 27110.739,E2 27110.739} C_VEL
LIN {X 0,Y 575.915,Z 846.786,A -85,B 0,C 180,E1 27109.257,E2 27109.257} C_VEL
LIN {X 0,Y 575.918,Z 845.092,A -85,B 0,C 180,E1 27107.789,E2 27107.789} C_VEL
LIN {X 0,Y 575.921,Z 841.581,A -85,B 0,C 180,E1 27106.332,E2 27106.332} C_VEL
LIN {X 0,Y 575.939,Z 836.67,A -85,B 0,C 180,E1 27104.989,E2 27104.989} C_VEL
LIN {X 0,Y 575.97,Z 829.298,A -85,B 0,C 180,E1 27103.551,E2 27103.551} C_VEL
LIN {X 0,Y 576.026,Z 820.974,A -85,B 0,C 180,E1 27102.325,E2 27102.325} C_VEL
LIN {X 0,Y 576.097,Z 811.27,A -85,B 0,C 180,E1 27101.207,E2 27101.207} C_VEL
LIN {X 0,Y 576.196,Z 800.248,A -85,B 0,C 180,E1 27100.193,E2 27100.193} C_VEL
LIN {X 0,Y 576.279,Z 788.31,A -85,B 0,C 180,E1 27099.334,E2 27099.334} C_VEL
LIN {X 0,Y 576.421,Z 774.585,A -85,B 0,C 180,E1 27098.577,E2 27098.577} C_VEL
LIN {X 0,Y 576.524,Z 759.821,A -85,B 0,C 180,E1 27097.993,E2 27097.993} C_VEL
LIN {X 0,Y 576.588,Z 745.002,A -85,B 0,C 180,E1 27097.612,E2 27097.612} C_VEL
LIN {X 0,Y 576.638,Z 699.18,A -85,B 0,C 180,E1 27097.009,E2 27097.009} C_VEL
LIN {X 0,Y 576.532,Z 634.266,A -85,B 0,C 180,E1 27096.193,E2 27096.193} C_VEL
LIN {X 0,Y 576.364,Z 632.451,A -85,B 0,C 180,E1 27096.123,E2 27096.123} C_VEL
LIN {X 0,Y 576.546,Z 601.609,A -85,B 0,C 180,E1 27092.881,E2 27092.881} C_VEL
LIN {X 0,Y 576.851,Z 571.017,A -85,B 0,C 180,E1 27089.602,E2 27089.602} C_VEL
LIN {X 0,Y 577.156,Z 541.055,A -85,B 0,C 180,E1 27086.324,E2 27086.324} C_VEL
LIN {X 0,Y 577.497,Z 512.632,A -85,B 0,C 180,E1 27083.138,E2 27083.138} C_VEL
LIN {X 0,Y 576.108,Z 507.191,A -85,B 0,C 180,E1 27082.395,E2 27082.395} C_VEL
LIN {X 0,Y 576.113,Z 507.036,A -85,B 0,C 180,E1 27079.196,E2 27079.196} C_VEL
LIN {X 0,Y 576.082,Z 507.032,A -85,B 0,C 180,E1 27076.244,E2 27076.244} C_VEL
LIN {X 0,Y 576.103,Z 507.033,A -85,B 0,C 180,E1 27072.944,E2 27072.944} C_VEL
LIN {X 0,Y 576.077,Z 507.032,A -85,B 0,C 180,E1 27070.112,E2 27070.112} C_VEL
LIN {X 0,Y 576.116,Z 507.025,A -85,B 0,C 180,E1 27066.901,E2 27066.901} C_VEL
LIN {X 0,Y 576.073,Z 507.033,A -85,B 0,C 180,E1 27063.953,E2 27063.953} C_VEL
LIN {X 0,Y 576.125,Z 507.027,A -85,B 0,C 180,E1 27060.804,E2 27060.804} C_VEL
LIN {X 0,Y 576.069,Z 507.029,A -85,B 0,C 180,E1 27057.804,E2 27057.804} C_VEL
LIN {X 0,Y 576.131,Z 507.032,A -85,B 0,C 180,E1 27054.654,E2 27054.654} C_VEL
LIN {X 0,Y 576.074,Z 507.032,A -85,B 0,C 180,E1 27051.587,E2 27051.587} C_VEL
LIN {X 0,Y 576.128,Z 507.03,A -85,B 0,C 180,E1 27048.417,E2 27048.417} C_VEL
LIN {X 0,Y 576.076,Z 507.032,A -85,B 0,C 180,E1 27045.48,E2 27045.48} C_VEL
LIN {X 0,Y 576.145,Z 507.028,A -85,B 0,C 180,E1 27042.326,E2 27042.326} C_VEL
LIN {X 0,Y 576.079,Z 507.031,A -85,B 0,C 180,E1 27039.282,E2 27039.282} C_VEL
LIN {X 0,Y 576.15,Z 507.029,A -85,B 0,C 180,E1 27036.16,E2 27036.16} C_VEL
LIN {X 0,Y 576.08,Z 507.029,A -85,B 0,C 180,E1 27033.143,E2 27033.143} C_VEL
LIN {X 0,Y 576.159,Z 507.03,A -85,B 0,C 180,E1 27029.987,E2 27029.987} C_VEL
LIN {X 0,Y 576.085,Z 507.029,A -85,B 0,C 180,E1 27026.868,E2 27026.868} C_VEL
LIN {X 0,Y 576.152,Z 507.029,A -85,B 0,C 180,E1 27023.742,E2 27023.742} C_VEL
LIN {X 0,Y 576.089,Z 507.031,A -85,B 0,C 180,E1 27020.63,E2 27020.63} C_VEL
LIN {X 0,Y 576.129,Z 507.025,A -85,B 0,C 180,E1 27017.36,E2 27017.36} C_VEL
LIN {X 0,Y 576.096,Z 507.031,A -85,B 0,C 180,E1 27014.371,E2 27014.371} C_VEL
LIN {X 0,Y 576.125,Z 507.027,A -85,B 0,C 180,E1 27011.107,E2 27011.107} C_VEL
LIN {X 0,Y 576.101,Z 507.026,A -85,B 0,C 180,E1 27008.082,E2 27008.082} C_VEL
LIN {X 0,Y 576.108,Z 507.029,A -85,B 0,C 180,E1 27004.679,E2 27004.679} C_VEL
LIN {X 0,Y 576.123,Z 507.03,A -85,B 0,C 180,E1 27001.664,E2 27001.664} C_VEL
LIN {X 0,Y 576.105,Z 507.028,A -85,B 0,C 180,E1 26998.4,E2 26998.4} C_VEL
LIN {X 0,Y 576.141,Z 507.033,A -85,B 0,C 180,E1 26995.322,E2 26995.322} C_VEL
LIN {X 0,Y 576.103,Z 507.025,A -85,B 0,C 180,E1 26992.12,E2 26992.12} C_VEL
LIN {X 0,Y 576.155,Z 507.034,A -85,B 0,C 180,E1 26988.995,E2 26988.995} C_VEL
LIN {X 0,Y 576.103,Z 507.026,A -85,B 0,C 180,E1 26985.835,E2 26985.835} C_VEL
LIN {X 0,Y 576.162,Z 507.029,A -85,B 0,C 180,E1 26982.634,E2 26982.634} C_VEL
LIN {X 0,Y 576.105,Z 507.028,A -85,B 0,C 180,E1 26979.477,E2 26979.477} C_VEL
LIN {X 0,Y 576.161,Z 507.026,A -85,B 0,C 180,E1 26976.259,E2 26976.259} C_VEL
LIN {X 0,Y 576.115,Z 507.028,A -85,B 0,C 180,E1 26973.066,E2 26973.066} C_VEL
LIN {X 0,Y 576.137,Z 507.025,A -85,B 0,C 180,E1 26969.783,E2 26969.783} C_VEL
LIN {X 0,Y 576.138,Z 507.032,A -85,B 0,C 180,E1 26966.585,E2 26966.585} C_VEL
LIN {X 0,Y 576.119,Z 507.027,A -85,B 0,C 180,E1 26963.298,E2 26963.298} C_VEL
LIN {X 0,Y 576.16,Z 507.031,A -85,B 0,C 180,E1 26960.085,E2 26960.085} C_VEL
LIN {X 0,Y 576.114,Z 507.029,A -85,B 0,C 180,E1 26956.859,E2 26956.859} C_VEL
LIN {X 0,Y 576.158,Z 507.027,A -85,B 0,C 180,E1 26953.643,E2 26953.643} C_VEL
LIN {X 0,Y 576.119,Z 507.031,A -85,B 0,C 180,E1 26950.47,E2 26950.47} C_VEL
LIN {X 0,Y 576.15,Z 507.026,A -85,B 0,C 180,E1 26947.149,E2 26947.149} C_VEL
LIN {X 0,Y 576.15,Z 507.034,A -85,B 0,C 180,E1 26943.851,E2 26943.851} C_VEL
LIN {X 0,Y 576.19,Z 507.27,A -85,B 0,C 180,E1 26941.312,E2 26941.312} C_VEL
LIN {X 0,Y 578.898,Z 515.991,A -85,B 0,C 180,E1 26940.474,E2 26940.474} C_VEL
LIN {X 0,Y 578.309,Z 559.528,A -85,B 0,C 180,E1 26937.379,E2 26937.379} C_VEL
LIN {X 0,Y 577.818,Z 604.159,A -85,B 0,C 180,E1 26934.283,E2 26934.283} C_VEL
LIN {X 0,Y 577.825,Z 615.273,A -85,B 0,C 180,E1 26933.556,E2 26933.556} C_VEL
LIN {X 0,Y 578.379,Z 621.348,A -85,B 0,C 180,E1 26933.448,E2 26933.448} C_VEL
LIN {X 0,Y 577.839,Z 824.35,A -85,B 0,C 180,E1 26930.776,E2 26930.776} C_VEL
LIN {X 0,Y 577.668,Z 843.369,A -85,B 0,C 180,E1 26930.335,E2 26930.335} C_VEL
LIN {X 0,Y 577.491,Z 861.417,A -85,B 0,C 180,E1 26929.731,E2 26929.731} C_VEL
LIN {X 0,Y 577.246,Z 879.422,A -85,B 0,C 180,E1 26928.932,E2 26928.932} C_VEL
LIN {X 0,Y 577.027,Z 896.598,A -85,B 0,C 180,E1 26927.965,E2 26927.965} C_VEL
LIN {X 0,Y 576.783,Z 912.973,A -85,B 0,C 180,E1 26926.828,E2 26926.828} C_VEL
LIN {X 0,Y 576.55,Z 928.225,A -85,B 0,C 180,E1 26925.541,E2 26925.541} C_VEL
LIN {X 0,Y 576.349,Z 942.169,A -85,B 0,C 180,E1 26924.126,E2 26924.126} C_VEL
LIN {X 0,Y 576.201,Z 954.458,A -85,B 0,C 180,E1 26922.629,E2 26922.629} C_VEL
LIN {X 0,Y 576.083,Z 965.502,A -85,B 0,C 180,E1 26921.007,E2 26921.007} C_VEL
LIN {X 0,Y 575.998,Z 975.022,A -85,B 0,C 180,E1 26919.291,E2 26919.291} C_VEL
LIN {X 0,Y 575.955,Z 982.581,A -85,B 0,C 180,E1 26917.582,E2 26917.582} C_VEL
LIN {X 0,Y 575.921,Z 988.711,A -85,B 0,C 180,E1 26915.78,E2 26915.78} C_VEL
LIN {X 0,Y 575.92,Z 993.078,A -85,B 0,C 180,E1 26913.983,E2 26913.983} C_VEL
LIN {X 0,Y 575.916,Z 995.9,A -85,B 0,C 180,E1 26912.09,E2 26912.09} C_VEL
LIN {X 0,Y 575.909,Z 996.961,A -85,B 0,C 180,E1 26910.2,E2 26910.2} C_VEL
LIN {X 0,Y 575.913,Z 996.282,A -85,B 0,C 180,E1 26908.31,E2 26908.31} C_VEL
LIN {X 0,Y 575.91,Z 993.848,A -85,B 0,C 180,E1 26906.418,E2 26906.418} C_VEL
LIN {X 0,Y 575.922,Z 989.594,A -85,B 0,C 180,E1 26904.522,E2 26904.522} C_VEL
LIN {X 0,Y 575.943,Z 983.768,A -85,B 0,C 180,E1 26902.721,E2 26902.721} C_VEL
LIN {X 0,Y 576.001,Z 976.05,A -85,B 0,C 180,E1 26900.913,E2 26900.913} C_VEL
LIN {X 0,Y 576.075,Z 966.784,A -85,B 0,C 180,E1 26899.198,E2 26899.198} C_VEL
LIN {X 0,Y 576.191,Z 956.018,A -85,B 0,C 180,E1 26897.576,E2 26897.576} C_VEL
LIN {X 0,Y 576.34,Z 943.746,A -85,B 0,C 180,E1 26896.048,E2 26896.048} C_VEL
LIN {X 0,Y 576.525,Z 930.13,A -85,B 0,C 180,E1 26894.636,E2 26894.636} C_VEL
LIN {X 0,Y 576.744,Z 914.992,A -85,B 0,C 180,E1 26893.329,E2 26893.329} C_VEL
LIN {X 0,Y 576.982,Z 899.059,A -85,B 0,C 180,E1 26892.193,E2 26892.193} C_VEL
LIN {X 0,Y 577.19,Z 882.112,A -85,B 0,C 180,E1 26891.207,E2 26891.207} C_VEL
LIN {X 0,Y 577.45,Z 864.045,A -85,B 0,C 180,E1 26890.375,E2 26890.375} C_VEL
LIN {X 0,Y 577.633,Z 845.408,A -85,B 0,C 180,E1 26889.725,E2 26889.725} C_VEL
LIN {X 0,Y 577.809,Z 826.751,A -85,B 0,C 180,E1 26889.272,E2 26889.272} C_VEL
LIN {X 0,Y 577.934,Z 797.626,A -85,B 0,C 180,E1 26888.852,E2 26888.852} C_VEL
LIN {X 0,Y 578.206,Z 617.786,A -85,B 0,C 180,E1 26886.497,E2 26886.497} C_VEL
LIN {X 0,Y 577.736,Z 613.94,A -85,B 0,C 180,E1 26886.385,E2 26886.385} C_VEL
LIN {X 0,Y 578.232,Z 566.733,A -85,B 0,C 180,E1 26883.126,E2 26883.126} C_VEL
LIN {X 0,Y 578.811,Z 522.55,A -85,B 0,C 180,E1 26879.998,E2 26879.998} C_VEL
LIN {X 0,Y 578.819,Z 515.034,A -85,B 0,C 180,E1 26879.452,E2 26879.452} C_VEL
LIN {X 0,Y 576.192,Z 507.283,A -85,B 0,C 180,E1 26878.691,E2 26878.691} C_VEL
LIN {X 0,Y 576.118,Z 507.032,A -85,B 0,C 180,E1 26875.549,E2 26875.549} C_VEL
LIN {X 0,Y 576.161,Z 507.031,A -85,B 0,C 180,E1 26872.31,E2 26872.31} C_VEL
LIN {X 0,Y 576.117,Z 507.028,A -85,B 0,C 180,E1 26869.14,E2 26869.14} C_VEL
LIN {X 0,Y 576.131,Z 507.033,A -85,B 0,C 180,E1 26865.787,E2 26865.787} C_VEL
LIN {X 0,Y 576.139,Z 507.028,A -85,B 0,C 180,E1 26862.596,E2 26862.596} C_VEL
LIN {X 0,Y 576.104,Z 507.029,A -85,B 0,C 180,E1 26859.307,E2 26859.307} C_VEL
LIN {X 0,Y 576.158,Z 507.029,A -85,B 0,C 180,E1 26856.159,E2 26856.159} C_VEL
LIN {X 0,Y 576.095,Z 507.031,A -85,B 0,C 180,E1 26853.023,E2 26853.023} C_VEL
LIN {X 0,Y 576.164,Z 507.031,A -85,B 0,C 180,E1 26849.82,E2 26849.82} C_VEL
LIN {X 0,Y 576.088,Z 507.031,A -85,B 0,C 180,E1 26846.713,E2 26846.713} C_VEL
LIN {X 0,Y 576.146,Z 507.032,A -85,B 0,C 180,E1 26843.525,E2 26843.525} C_VEL
LIN {X 0,Y 576.081,Z 507.032,A -85,B 0,C 180,E1 26840.524,E2 26840.524} C_VEL
LIN {X 0,Y 576.139,Z 507.034,A -85,B 0,C 180,E1 26837.367,E2 26837.367} C_VEL
LIN {X 0,Y 576.072,Z 507.03,A -85,B 0,C 180,E1 26834.371,E2 26834.371} C_VEL
LIN {X 0,Y 576.133,Z 507.032,A -85,B 0,C 180,E1 26831.208,E2 26831.208} C_VEL
LIN {X 0,Y 576.072,Z 507.033,A -85,B 0,C 180,E1 26828.182,E2 26828.182} C_VEL
LIN {X 0,Y 576.143,Z 507.029,A -85,B 0,C 180,E1 26825.078,E2 26825.078} C_VEL
LIN {X 0,Y 576.081,Z 507.033,A -85,B 0,C 180,E1 26821.989,E2 26821.989} C_VEL
LIN {X 0,Y 576.137,Z 507.03,A -85,B 0,C 180,E1 26818.807,E2 26818.807} C_VEL
LIN {X 0,Y 576.092,Z 507.031,A -85,B 0,C 180,E1 26815.72,E2 26815.72} C_VEL
LIN {X 0,Y 576.119,Z 507.029,A -85,B 0,C 180,E1 26812.42,E2 26812.42} C_VEL
LIN {X 0,Y 576.107,Z 507.031,A -85,B 0,C 180,E1 26809.399,E2 26809.399} C_VEL
LIN {X 0,Y 576.108,Z 507.028,A -85,B 0,C 180,E1 26806.04,E2 26806.04} C_VEL
LIN {X 0,Y 576.116,Z 507.032,A -85,B 0,C 180,E1 26803.216,E2 26803.216} C_VEL
LIN {X 0,Y 575.163,Z 507.157,A -85,B 0,C 180,E1 26802.45,E2 26802.45} C_VEL
LIN {X 0,Y 568.623,Z 507.965,A -85,B 0,C 180,E1 26800.244,E2 26800.244} C_VEL
LIN {X 0,Y 568.169,Z 508.018,A -85,B 0,C 180,E1 26799.739,E2 26799.739} C_VEL
LIN {X 0,Y 568.224,Z 508.018,A -85,B 0,C 180,E1 26796.567,E2 26796.567} C_VEL
LIN {X 0,Y 568.171,Z 508.019,A -85,B 0,C 180,E1 26793.336,E2 26793.336} C_VEL
LIN {X 0,Y 568.222,Z 508.016,A -85,B 0,C 180,E1 26790.134,E2 26790.134} C_VEL
LIN {X 0,Y 568.187,Z 508.021,A -85,B 0,C 180,E1 26786.881,E2 26786.881} C_VEL
LIN {X 0,Y 568.196,Z 508.017,A -85,B 0,C 180,E1 26783.503,E2 26783.503} C_VEL
LIN {X 0,Y 568.219,Z 508.021,A -85,B 0,C 180,E1 26780.253,E2 26780.253} C_VEL
LIN {X 0,Y 568.249,Z 508.248,A -85,B 0,C 180,E1 26777.834,E2 26777.834} C_VEL
LIN {X 0,Y 569.996,Z 515.757,A -85,B 0,C 180,E1 26776.833,E2 26776.833} C_VEL
LIN {X 0,Y 569.458,Z 544.343,A -85,B 0,C 180,E1 26773.555,E2 26773.555} C_VEL
LIN {X 0,Y 569.062,Z 574.528,A -85,B 0,C 180,E1 26770.213,E2 26770.213} C_VEL
LIN {X 0,Y 568.719,Z 605.266,A -85,B 0,C 180,E1 26766.876,E2 26766.876} C_VEL
LIN {X 0,Y 568.475,Z 632.957,A -85,B 0,C 180,E1 26763.948,E2 26763.948} C_VEL
LIN {X 0,Y 568.986,Z 639.612,A -85,B 0,C 180,E1 26763.835,E2 26763.835} C_VEL
LIN {X 0,Y 568.739,Z 744.358,A -85,B 0,C 180,E1 26762.484,E2 26762.484} C_VEL
LIN {X 0,Y 568.684,Z 759.484,A -85,B 0,C 180,E1 26762.097,E2 26762.097} C_VEL
LIN {X 0,Y 568.562,Z 773.52,A -85,B 0,C 180,E1 26761.541,E2 26761.541} C_VEL
LIN {X 0,Y 568.412,Z 786.167,A -85,B 0,C 180,E1 26760.861,E2 26760.861} C_VEL
LIN {X 0,Y 568.275,Z 798.782,A -85,B 0,C 180,E1 26759.975,E2 26759.975} C_VEL
LIN {X 0,Y 568.161,Z 810.214,A -85,B 0,C 180,E1 26758.939,E2 26758.939} C_VEL
LIN {X 0,Y 568.064,Z 820.166,A -85,B 0,C 180,E1 26757.799,E2 26757.799} C_VEL
LIN {X 0,Y 567.988,Z 828.676,A -85,B 0,C 180,E1 26756.556,E2 26756.556} C_VEL
LIN {X 0,Y 567.947,Z 835.77,A -85,B 0,C 180,E1 26755.191,E2 26755.191} C_VEL
LIN {X 0,Y 567.925,Z 841.151,A -85,B 0,C 180,E1 26753.773,E2 26753.773} C_VEL
LIN {X 0,Y 567.917,Z 844.942,A -85,B 0,C 180,E1 26752.239,E2 26752.239} C_VEL
LIN {X 0,Y 567.918,Z 846.747,A -85,B 0,C 180,E1 26750.721,E2 26750.721} C_VEL
LIN {X 0,Y 567.915,Z 846.767,A -85,B 0,C 180,E1 26749.219,E2 26749.219} C_VEL
LIN {X 0,Y 567.917,Z 845.046,A -85,B 0,C 180,E1 26747.73,E2 26747.73} C_VEL
LIN {X 0,Y 567.923,Z 841.499,A -85,B 0,C 180,E1 26746.253,E2 26746.253} C_VEL
LIN {X 0,Y 567.944,Z 836.45,A -85,B 0,C 180,E1 26744.869,E2 26744.869} C_VEL
LIN {X 0,Y 567.986,Z 829.147,A -85,B 0,C 180,E1 26743.434,E2 26743.434} C_VEL
LIN {X 0,Y 568.058,Z 820.774,A -85,B 0,C 180,E1 26742.191,E2 26742.191} C_VEL
LIN {X 0,Y 568.15,Z 811.034,A -85,B 0,C 180,E1 26741.057,E2 26741.057} C_VEL
LIN {X 0,Y 568.278,Z 799.933,A -85,B 0,C 180,E1 26740.029,E2 26740.029} C_VEL
LIN {X 0,Y 568.391,Z 787.897,A -85,B 0,C 180,E1 26739.158,E2 26739.158} C_VEL
LIN {X 0,Y 568.552,Z 775.1,A -85,B 0,C 180,E1 26738.442,E2 26738.442} C_VEL
LIN {X 0,Y 568.677,Z 760.683,A -85,B 0,C 180,E1 26737.855,E2 26737.855} C_VEL
LIN {X 0,Y 568.767,Z 746.196,A -85,B 0,C 180,E1 26737.463,E2 26737.463} C_VEL
LIN {X 0,Y 568.812,Z 720.309,A -85,B 0,C 180,E1 26737.096,E2 26737.096} C_VEL
LIN {X 0,Y 568.766,Z 635.104,A -85,B 0,C 180,E1 26736.012,E2 26736.012} C_VEL
LIN {X 0,Y 568.5,Z 632.828,A -85,B 0,C 180,E1 26735.954,E2 26735.954} C_VEL
LIN {X 0,Y 568.716,Z 603.285,A -85,B 0,C 180,E1 26732.82,E2 26732.82} C_VEL
LIN {X 0,Y 569.09,Z 572.687,A -85,B 0,C 180,E1 26729.495,E2 26729.495} C_VEL
LIN {X 0,Y 569.478,Z 542.722,A -85,B 0,C 180,E1 26726.174,E2 26726.174} C_VEL
LIN {X 0,Y 569.959,Z 515.14,A -85,B 0,C 180,E1 26723.022,E2 26723.022} C_VEL
LIN {X 0,Y 568.192,Z 508.144,A -85,B 0,C 180,E1 26722.059,E2 26722.059} C_VEL
LIN {X 0,Y 568.146,Z 508.025,A -85,B 0,C 180,E1 26718.838,E2 26718.838} C_VEL
LIN {X 0,Y 568.175,Z 508.021,A -85,B 0,C 180,E1 26715.841,E2 26715.841} C_VEL
LIN {X 0,Y 568.14,Z 508.022,A -85,B 0,C 180,E1 26712.592,E2 26712.592} C_VEL
LIN {X 0,Y 568.178,Z 508.021,A -85,B 0,C 180,E1 26709.609,E2 26709.609} C_VEL
LIN {X 0,Y 568.138,Z 508.012,A -85,B 0,C 180,E1 26706.454,E2 26706.454} C_VEL
LIN {X 0,Y 568.17,Z 508.022,A -85,B 0,C 180,E1 26703.451,E2 26703.451} C_VEL
LIN {X 0,Y 568.132,Z 508.014,A -85,B 0,C 180,E1 26700.186,E2 26700.186} C_VEL
LIN {X 0,Y 568.178,Z 508.018,A -85,B 0,C 180,E1 26697.181,E2 26697.181} C_VEL
LIN {X 0,Y 568.135,Z 508.021,A -85,B 0,C 180,E1 26694.001,E2 26694.001} C_VEL
LIN {X 0,Y 568.195,Z 508.021,A -85,B 0,C 180,E1 26690.899,E2 26690.899} C_VEL
LIN {X 0,Y 568.136,Z 508.018,A -85,B 0,C 180,E1 26687.76,E2 26687.76} C_VEL
LIN {X 0,Y 568.2,Z 508.022,A -85,B 0,C 180,E1 26684.694,E2 26684.694} C_VEL
LIN {X 0,Y 568.14,Z 508.017,A -85,B 0,C 180,E1 26681.566,E2 26681.566} C_VEL
LIN {X 0,Y 568.2,Z 508.021,A -85,B 0,C 180,E1 26678.531,E2 26678.531} C_VEL
LIN {X 0,Y 568.144,Z 508.018,A -85,B 0,C 180,E1 26675.38,E2 26675.38} C_VEL
LIN {X 0,Y 568.201,Z 508.018,A -85,B 0,C 180,E1 26672.341,E2 26672.341} C_VEL
LIN {X 0,Y 568.145,Z 508.02,A -85,B 0,C 180,E1 26669.176,E2 26669.176} C_VEL
LIN {X 0,Y 568.211,Z 508.016,A -85,B 0,C 180,E1 26666.099,E2 26666.099} C_VEL
LIN {X 0,Y 568.147,Z 508.02,A -85,B 0,C 180,E1 26662.888,E2 26662.888} C_VEL
LIN {X 0,Y 568.219,Z 508.016,A -85,B 0,C 180,E1 26659.721,E2 26659.721} C_VEL
LIN {X 0,Y 568.15,Z 508.015,A -85,B 0,C 180,E1 26656.565,E2 26656.565} C_VEL
LIN {X 0,Y 568.205,Z 508.018,A -85,B 0,C 180,E1 26653.335,E2 26653.335} C_VEL
LIN {X 0,Y 568.158,Z 508.018,A -85,B 0,C 180,E1 26650.239,E2 26650.239} C_VEL
LIN {X 0,Y 568.178,Z 508.016,A -85,B 0,C 180,E1 26646.873,E2 26646.873} C_VEL
LIN {X 0,Y 568.175,Z 508.021,A -85,B 0,C 180,E1 26643.835,E2 26643.835} C_VEL
LIN {X 0,Y 568.167,Z 508.011,A -85,B 0,C 180,E1 26640.504,E2 26640.504} C_VEL
LIN {X 0,Y 568.191,Z 508.02,A -85,B 0,C 180,E1 26637.479,E2 26637.479} C_VEL
LIN {X 0,Y 568.166,Z 508.016,A -85,B 0,C 180,E1 26634.243,E2 26634.243} C_VEL
LIN {X 0,Y 568.214,Z 508.017,A -85,B 0,C 180,E1 26631.092,E2 26631.092} C_VEL
LIN {X 0,Y 568.164,Z 508.018,A -85,B 0,C 180,E1 26627.809,E2 26627.809} C_VEL
LIN {X 0,Y 568.223,Z 508.015,A -85,B 0,C 180,E1 26624.591,E2 26624.591} C_VEL
LIN {X 0,Y 568.169,Z 508.019,A -85,B 0,C 180,E1 26621.427,E2 26621.427} C_VEL
LIN {X 0,Y 568.201,Z 508.014,A -85,B 0,C 180,E1 26618.096,E2 26618.096} C_VEL
LIN {X 0,Y 568.19,Z 508.021,A -85,B 0,C 180,E1 26614.907,E2 26614.907} C_VEL
LIN {X 0,Y 568.18,Z 508.016,A -85,B 0,C 180,E1 26611.621,E2 26611.621} C_VEL
LIN {X 0,Y 568.214,Z 508.019,A -85,B 0,C 180,E1 26608.492,E2 26608.492} C_VEL
LIN {X 0,Y 568.173,Z 508.017,A -85,B 0,C 180,E1 26605.238,E2 26605.238} C_VEL
LIN {X 0,Y 568.221,Z 508.016,A -85,B 0,C 180,E1 26602.024,E2 26602.024} C_VEL
LIN {X 0,Y 568.176,Z 508.019,A -85,B 0,C 180,E1 26598.841,E2 26598.841} C_VEL
LIN {X 0,Y 568.22,Z 508.013,A -85,B 0,C 180,E1 26595.546,E2 26595.546} C_VEL
LIN {X 0,Y 568.197,Z 508.021,A -85,B 0,C 180,E1 26592.235,E2 26592.235} C_VEL
LIN {X 0,Y 568.19,Z 508.016,A -85,B 0,C 180,E1 26588.917,E2 26588.917} C_VEL
LIN {X 0,Y 568.22,Z 508.02,A -85,B 0,C 180,E1 26585.615,E2 26585.615} C_VEL
LIN {X 0,Y 568.18,Z 508.013,A -85,B 0,C 180,E1 26582.34,E2 26582.34} C_VEL
LIN {X 0,Y 568.257,Z 508.295,A -85,B 0,C 180,E1 26581.692,E2 26581.692} C_VEL
LIN {X 0,Y 571.665,Z 518.574,A -85,B 0,C 180,E1 26580.71,E2 26580.71} C_VEL
LIN {X 0,Y 570.937,Z 561.68,A -85,B 0,C 180,E1 26577.608,E2 26577.608} C_VEL
LIN {X 0,Y 570.306,Z 606.782,A -85,B 0,C 180,E1 26574.44,E2 26574.44} C_VEL
LIN {X 0,Y 570.318,Z 615.28,A -85,B 0,C 180,E1 26573.885,E2 26573.885} C_VEL
LIN {X 0,Y 571.038,Z 621.984,A -85,B 0,C 180,E1 26573.759,E2 26573.759} C_VEL
LIN {X 0,Y 570.356,Z 824.35,A -85,B 0,C 180,E1 26571.061,E2 26571.061} C_VEL
LIN {X 0,Y 570.148,Z 843.368,A -85,B 0,C 180,E1 26570.616,E2 26570.616} C_VEL
LIN {X 0,Y 569.92,Z 861.415,A -85,B 0,C 180,E1 26570.005,E2 26570.005} C_VEL
LIN {X 0,Y 569.624,Z 879.249,A -85,B 0,C 180,E1 26569.205,E2 26569.205} C_VEL
LIN {X 0,Y 569.349,Z 895.784,A -85,B 0,C 180,E1 26568.268,E2 26568.268} C_VEL
LIN {X 0,Y 569.054,Z 911.635,A -85,B 0,C 180,E1 26567.168,E2 26567.168} C_VEL
LIN {X 0,Y 568.768,Z 926.561,A -85,B 0,C 180,E1 26565.916,E2 26565.916} C_VEL
LIN {X 0,Y 568.523,Z 940.02,A -85,B 0,C 180,E1 26564.566,E2 26564.566} C_VEL
LIN {X 0,Y 568.307,Z 952.911,A -85,B 0,C 180,E1 26563.015,E2 26563.015} C_VEL
LIN {X 0,Y 568.142,Z 964.228,A -85,B 0,C 180,E1 26561.368,E2 26561.368} C_VEL
LIN {X 0,Y 568.032,Z 973.992,A -85,B 0,C 180,E1 26559.627,E2 26559.627} C_VEL
LIN {X 0,Y 567.964,Z 981.771,A -85,B 0,C 180,E1 26557.893,E2 26557.893} C_VEL
LIN {X 0,Y 567.932,Z 988.107,A -85,B 0,C 180,E1 26556.064,E2 26556.064} C_VEL
LIN {X 0,Y 567.92,Z 992.874,A -85,B 0,C 180,E1 26554.14,E2 26554.14} C_VEL
LIN {X 0,Y 567.916,Z 995.789,A -85,B 0,C 180,E1 26552.221,E2 26552.221} C_VEL
LIN {X 0,Y 567.907,Z 996.939,A -85,B 0,C 180,E1 26550.304,E2 26550.304} C_VEL
LIN {X 0,Y 567.914,Z 996.349,A -85,B 0,C 180,E1 26548.387,E2 26548.387} C_VEL
LIN {X 0,Y 567.909,Z 994.007,A -85,B 0,C 180,E1 26546.469,E2 26546.469} C_VEL
LIN {X 0,Y 567.923,Z 990.102,A -85,B 0,C 180,E1 26544.648,E2 26544.648} C_VEL
LIN {X 0,Y 567.946,Z 984.475,A -85,B 0,C 180,E1 26542.821,E2 26542.821} C_VEL
LIN {X 0,Y 568,Z 977.434,A -85,B 0,C 180,E1 26541.091,E2 26541.091} C_VEL
LIN {X 0,Y 568.096,Z 968.526,A -85,B 0,C 180,E1 26539.353,E2 26539.353} C_VEL
LIN {X 0,Y 568.231,Z 958.165,A -85,B 0,C 180,E1 26537.709,E2 26537.709} C_VEL
LIN {X 0,Y 568.412,Z 946.369,A -85,B 0,C 180,E1 26536.161,E2 26536.161} C_VEL
LIN {X 0,Y 568.647,Z 933.109,A -85,B 0,C 180,E1 26534.71,E2 26534.71} C_VEL
LIN {X 0,Y 568.927,Z 918.259,A -85,B 0,C 180,E1 26533.356,E2 26533.356} C_VEL
LIN {X 0,Y 569.234,Z 902.273,A -85,B 0,C 180,E1 26532.154,E2 26532.154} C_VEL
LIN {X 0,Y 569.511,Z 885.198,A -85,B 0,C 180,E1 26531.108,E2 26531.108} C_VEL
LIN {X 0,Y 569.833,Z 867.874,A -85,B 0,C 180,E1 26530.262,E2 26530.262} C_VEL
LIN {X 0,Y 570.07,Z 849.731,A -85,B 0,C 180,E1 26529.578,E2 26529.578} C_VEL
LIN {X 0,Y 570.291,Z 831.133,A -85,B 0,C 180,E1 26529.077,E2 26529.077} C_VEL
LIN {X 0,Y 570.432,Z 811.063,A -85,B 0,C 180,E1 26528.738,E2 26528.738} C_VEL
LIN {X 0,Y 570.879,Z 618.938,A -85,B 0,C 180,E1 26526.193,E2 26526.193} C_VEL
LIN {X 0,Y 570.231,Z 613.94,A -85,B 0,C 180,E1 26526.055,E2 26526.055} C_VEL
LIN {X 0,Y 570.865,Z 566.654,A -85,B 0,C 180,E1 26522.745,E2 26522.745} C_VEL
LIN {X 0,Y 571.597,Z 522.611,A -85,B 0,C 180,E1 26519.584,E2 26519.584} C_VEL
LIN {X 0,Y 571.477,Z 517.654,A -85,B 0,C 180,E1 26519.211,E2 26519.211} C_VEL
LIN {X 0,Y 568.269,Z 508.361,A -85,B 0,C 180,E1 26518.323,E2 26518.323} C_VEL
LIN {X 0,Y 568.181,Z 508.017,A -85,B 0,C 180,E1 26517.638,E2 26517.638} C_VEL
LIN {X 0,Y 568.222,Z 508.02,A -85,B 0,C 180,E1 26514.383,E2 26514.383} C_VEL
LIN {X 0,Y 568.179,Z 508.017,A -85,B 0,C 180,E1 26511.215,E2 26511.215} C_VEL
LIN {X 0,Y 568.198,Z 508.022,A -85,B 0,C 180,E1 26507.905,E2 26507.905} C_VEL
LIN {X 0,Y 568.199,Z 508.016,A -85,B 0,C 180,E1 26504.697,E2 26504.697} C_VEL
LIN {X 0,Y 568.17,Z 508.02,A -85,B 0,C 180,E1 26501.428,E2 26501.428} C_VEL
LIN {X 0,Y 568.215,Z 508.015,A -85,B 0,C 180,E1 26498.272,E2 26498.272} C_VEL
LIN {X 0,Y 568.158,Z 508.019,A -85,B 0,C 180,E1 26495.092,E2 26495.092} C_VEL
LIN {X 0,Y 568.222,Z 508.018,A -85,B 0,C 180,E1 26491.982,E2 26491.982} C_VEL
LIN {X 0,Y 568.15,Z 508.019,A -85,B 0,C 180,E1 26488.829,E2 26488.829} C_VEL
LIN {X 0,Y 568.216,Z 508.022,A -85,B 0,C 180,E1 26485.65,E2 26485.65} C_VEL
LIN {X 0,Y 568.147,Z 508.02,A -85,B 0,C 180,E1 26482.508,E2 26482.508} C_VEL
LIN {X 0,Y 568.189,Z 508.02,A -85,B 0,C 180,E1 26479.319,E2 26479.319} C_VEL
LIN {X 0,Y 568.139,Z 508.022,A -85,B 0,C 180,E1 26476.354,E2 26476.354} C_VEL
LIN {X 0,Y 568.177,Z 508.023,A -85,B 0,C 180,E1 26473.121,E2 26473.121} C_VEL
LIN {X 0,Y 568.135,Z 508.021,A -85,B 0,C 180,E1 26470.136,E2 26470.136} C_VEL
LIN {X 0,Y 568.169,Z 508.022,A -85,B 0,C 180,E1 26466.873,E2 26466.873} C_VEL
LIN {X 0,Y 568.143,Z 508.019,A -85,B 0,C 180,E1 26463.935,E2 26463.935} C_VEL
LIN {X 0,Y 568.167,Z 508.017,A -85,B 0,C 180,E1 26460.605,E2 26460.605} C_VEL
LIN {X 0,Y 568.155,Z 508.021,A -85,B 0,C 180,E1 26457.68,E2 26457.68} C_VEL
LIN {X 0,Y 568.159,Z 508.019,A -85,B 0,C 180,E1 26454.243,E2 26454.243} C_VEL
LIN {X 0,Y 568.19,Z 508.022,A -85,B 0,C 180,E1 26451.193,E2 26451.193} C_VEL
LIN {X 0,Y 568.16,Z 508.019,A -85,B 0,C 180,E1 26447.911,E2 26447.911} C_VEL
LIN {X 0,Y 568.22,Z 508.022,A -85,B 0,C 180,E1 26444.8,E2 26444.8} C_VEL
LIN {X 0,Y 568.163,Z 508.018,A -85,B 0,C 180,E1 26441.639,E2 26441.639} C_VEL
LIN {X 0,Y 568.169,Z 508.018,A -85,B 0,C 180,E1 26439.739,E2 26439.739} C_VEL
LIN {X 0,Y 567.178,Z 508.148,A -85,B 0,C 180,E1 26438.963,E2 26438.963} C_VEL
LIN {X 0,Y 560.726,Z 508.955,A -85,B 0,C 180,E1 26436.726,E2 26436.726} C_VEL
LIN {X 0,Y 560.28,Z 509.002,A -85,B 0,C 180,E1 26436.214,E2 26436.214} C_VEL
LIN {X 0,Y 560.248,Z 509.01,A -85,B 0,C 180,E1 26432.929,E2 26432.929} C_VEL
LIN {X 0,Y 560.244,Z 509.007,A -85,B 0,C 180,E1 26429.531,E2 26429.531} C_VEL
LIN {X 0,Y 560.281,Z 509.008,A -85,B 0,C 180,E1 26426.254,E2 26426.254} C_VEL
LIN {X 0,Y 560.244,Z 509.01,A -85,B 0,C 180,E1 26423.027,E2 26423.027} C_VEL
LIN {X 0,Y 560.283,Z 509.007,A -85,B 0,C 180,E1 26419.758,E2 26419.758} C_VEL
LIN {X 0,Y 560.302,Z 509.166,A -85,B 0,C 180,E1 26418.201,E2 26418.201} C_VEL
LIN {X 0,Y 562.471,Z 518.583,A -85,B 0,C 180,E1 26416.93,E2 26416.93} C_VEL
LIN {X 0,Y 561.77,Z 547.23,A -85,B 0,C 180,E1 26413.581,E2 26413.581} C_VEL
LIN {X 0,Y 561.29,Z 577.067,A -85,B 0,C 180,E1 26410.222,E2 26410.222} C_VEL
LIN {X 0,Y 560.867,Z 607.933,A -85,B 0,C 180,E1 26406.828,E2 26406.828} C_VEL
LIN {X 0,Y 560.602,Z 633.055,A -85,B 0,C 180,E1 26404.144,E2 26404.144} C_VEL
LIN {X 0,Y 561.219,Z 640.144,A -85,B 0,C 180,E1 26404.025,E2 26404.025} C_VEL
LIN {X 0,Y 560.926,Z 744.461,A -85,B 0,C 180,E1 26402.659,E2 26402.659} C_VEL
LIN {X 0,Y 560.855,Z 759.124,A -85,B 0,C 180,E1 26402.281,E2 26402.281} C_VEL
LIN {X 0,Y 560.702,Z 773.827,A -85,B 0,C 180,E1 26401.692,E2 26401.692} C_VEL
LIN {X 0,Y 560.516,Z 786.911,A -85,B 0,C 180,E1 26400.968,E2 26400.968} C_VEL
LIN {X 0,Y 560.353,Z 799.372,A -85,B 0,C 180,E1 26400.07,E2 26400.07} C_VEL
LIN {X 0,Y 560.211,Z 810.789,A -85,B 0,C 180,E1 26399.008,E2 26399.008} C_VEL
LIN {X 0,Y 560.092,Z 820.664,A -85,B 0,C 180,E1 26397.845,E2 26397.845} C_VEL
LIN {X 0,Y 560.001,Z 829.24,A -85,B 0,C 180,E1 26396.553,E2 26396.553} C_VEL
LIN {X 0,Y 559.952,Z 836.357,A -85,B 0,C 180,E1 26395.134,E2 26395.134} C_VEL
LIN {X 0,Y 559.926,Z 841.568,A -85,B 0,C 180,E1 26393.686,E2 26393.686} C_VEL
LIN {X 0,Y 559.918,Z 844.995,A -85,B 0,C 180,E1 26392.242,E2 26392.242} C_VEL
LIN {X 0,Y 559.919,Z 846.837,A -85,B 0,C 180,E1 26390.593,E2 26390.593} C_VEL
LIN {X 0,Y 559.915,Z 846.678,A -85,B 0,C 180,E1 26389.071,E2 26389.071} C_VEL
LIN {X 0,Y 559.917,Z 844.792,A -85,B 0,C 180,E1 26387.562,E2 26387.562} C_VEL
LIN {X 0,Y 559.927,Z 841.1,A -85,B 0,C 180,E1 26386.066,E2 26386.066} C_VEL
LIN {X 0,Y 559.952,Z 835.955,A -85,B 0,C 180,E1 26384.686,E2 26384.686} C_VEL
LIN {X 0,Y 560.003,Z 828.995,A -85,B 0,C 180,E1 26383.314,E2 26383.314} C_VEL
LIN {X 0,Y 560.102,Z 819.789,A -85,B 0,C 180,E1 26381.949,E2 26381.949} C_VEL
LIN {X 0,Y 560.225,Z 809.802,A -85,B 0,C 180,E1 26380.799,E2 26380.799} C_VEL
LIN {X 0,Y 560.375,Z 798.336,A -85,B 0,C 180,E1 26379.757,E2 26379.757} C_VEL
LIN {X 0,Y 560.554,Z 784.987,A -85,B 0,C 180,E1 26378.82,E2 26378.82} C_VEL
LIN {X 0,Y 560.733,Z 771.17,A -85,B 0,C 180,E1 26378.096,E2 26378.096} C_VEL
LIN {X 0,Y 560.875,Z 757.043,A -85,B 0,C 180,E1 26377.566,E2 26377.566} C_VEL
LIN {X 0,Y 560.978,Z 741.96,A -85,B 0,C 180,E1 26377.204,E2 26377.204} C_VEL
LIN {X 0,Y 561.003,Z 635.897,A -85,B 0,C 180,E1 26375.825,E2 26375.825} C_VEL
LIN {X 0,Y 560.615,Z 632.5,A -85,B 0,C 180,E1 26375.73,E2 26375.73} C_VEL
LIN {X 0,Y 560.901,Z 602.162,A -85,B 0,C 180,E1 26372.451,E2 26372.451} C_VEL
LIN {X 0,Y 561.357,Z 571.611,A -85,B 0,C 180,E1 26369.08,E2 26369.08} C_VEL
LIN {X 0,Y 561.847,Z 542.71,A -85,B 0,C 180,E1 26365.815,E2 26365.815} C_VEL
LIN {X 0,Y 562.415,Z 517.652,A -85,B 0,C 180,E1 26362.902,E2 26362.902} C_VEL
LIN {X 0,Y 560.289,Z 509.105,A -85,B 0,C 180,E1 26361.714,E2 26361.714} C_VEL
LIN {X 0,Y 560.202,Z 509.014,A -85,B 0,C 180,E1 26358.485,E2 26358.485} C_VEL
LIN {X 0,Y 560.263,Z 509.011,A -85,B 0,C 180,E1 26355.301,E2 26355.301} C_VEL
LIN {X 0,Y 560.199,Z 509.011,A -85,B 0,C 180,E1 26352.23,E2 26352.23} C_VEL
LIN {X 0,Y 560.242,Z 509.011,A -85,B 0,C 180,E1 26348.971,E2 26348.971} C_VEL
LIN {X 0,Y 560.197,Z 508.999,A -85,B 0,C 180,E1 26345.988,E2 26345.988} C_VEL
LIN {X 0,Y 560.227,Z 509.011,A -85,B 0,C 180,E1 26342.699,E2 26342.699} C_VEL
LIN {X 0,Y 560.2,Z 509.002,A -85,B 0,C 180,E1 26339.663,E2 26339.663} C_VEL
LIN {X 0,Y 560.206,Z 509.011,A -85,B 0,C 180,E1 26336.276,E2 26336.276} C_VEL
LIN {X 0,Y 560.219,Z 509.01,A -85,B 0,C 180,E1 26333.261,E2 26333.261} C_VEL
LIN {X 0,Y 560.202,Z 509.011,A -85,B 0,C 180,E1 26329.969,E2 26329.969} C_VEL
LIN {X 0,Y 560.226,Z 509.007,A -85,B 0,C 180,E1 26327.021,E2 26327.021} C_VEL
LIN {X 0,Y 560.202,Z 509.01,A -85,B 0,C 180,E1 26323.713,E2 26323.713} C_VEL
LIN {X 0,Y 560.251,Z 509.006,A -85,B 0,C 180,E1 26320.648,E2 26320.648} C_VEL
LIN {X 0,Y 560.202,Z 509.01,A -85,B 0,C 180,E1 26317.421,E2 26317.421} C_VEL
LIN {X 0,Y 560.282,Z 509.003,A -85,B 0,C 180,E1 26314.204,E2 26314.204} C_VEL
LIN {X 0,Y 560.205,Z 509.009,A -85,B 0,C 180,E1 26311.052,E2 26311.052} C_VEL
LIN {X 0,Y 560.272,Z 509.003,A -85,B 0,C 180,E1 26307.877,E2 26307.877} C_VEL
LIN {X 0,Y 560.212,Z 509.005,A -85,B 0,C 180,E1 26304.715,E2 26304.715} C_VEL
LIN {X 0,Y 560.248,Z 509.007,A -85,B 0,C 180,E1 26301.461,E2 26301.461} C_VEL
LIN {X 0,Y 560.219,Z 509.005,A -85,B 0,C 180,E1 26298.416,E2 26298.416} C_VEL
LIN {X 0,Y 560.225,Z 509.007,A -85,B 0,C 180,E1 26294.998,E2 26294.998} C_VEL
LIN {X 0,Y 560.245,Z 509.01,A -85,B 0,C 180,E1 26291.948,E2 26291.948} C_VEL
LIN {X 0,Y 560.218,Z 509,A -85,B 0,C 180,E1 26288.623,E2 26288.623} C_VEL
LIN {X 0,Y 560.27,Z 509.009,A -85,B 0,C 180,E1 26285.53,E2 26285.53} C_VEL
LIN {X 0,Y 560.22,Z 509.005,A -85,B 0,C 180,E1 26282.353,E2 26282.353} C_VEL
LIN {X 0,Y 560.286,Z 509.005,A -85,B 0,C 180,E1 26279.182,E2 26279.182} C_VEL
LIN {X 0,Y 560.221,Z 509.008,A -85,B 0,C 180,E1 26276.009,E2 26276.009} C_VEL
LIN {X 0,Y 560.277,Z 508.998,A -85,B 0,C 180,E1 26272.721,E2 26272.721} C_VEL
LIN {X 0,Y 560.234,Z 509.008,A -85,B 0,C 180,E1 26269.512,E2 26269.512} C_VEL
LIN {X 0,Y 560.234,Z 509.002,A -85,B 0,C 180,E1 26266.058,E2 26266.058} C_VEL
LIN {X 0,Y 560.275,Z 509.01,A -85,B 0,C 180,E1 26262.875,E2 26262.875} C_VEL
LIN {X 0,Y 560.228,Z 509.004,A -85,B 0,C 180,E1 26259.634,E2 26259.634} C_VEL
LIN {X 0,Y 560.285,Z 509.007,A -85,B 0,C 180,E1 26256.438,E2 26256.438} C_VEL
LIN {X 0,Y 560.235,Z 509.004,A -85,B 0,C 180,E1 26253.158,E2 26253.158} C_VEL
LIN {X 0,Y 560.273,Z 509.002,A -85,B 0,C 180,E1 26249.903,E2 26249.903} C_VEL
LIN {X 0,Y 560.256,Z 509.01,A -85,B 0,C 180,E1 26246.633,E2 26246.633} C_VEL
LIN {X 0,Y 560.24,Z 509.006,A -85,B 0,C 180,E1 26243.253,E2 26243.253} C_VEL
LIN {X 0,Y 560.282,Z 509.009,A -85,B 0,C 180,E1 26240.026,E2 26240.026} C_VEL
LIN {X 0,Y 560.239,Z 509.008,A -85,B 0,C 180,E1 26236.729,E2 26236.729} C_VEL
LIN {X 0,Y 560.276,Z 509.003,A -85,B 0,C 180,E1 26233.395,E2 26233.395} C_VEL
LIN {X 0,Y 560.27,Z 509.009,A -85,B 0,C 180,E1 26230.04,E2 26230.04} C_VEL
LIN {X 0,Y 560.245,Z 509.007,A -85,B 0,C 180,E1 26226.715,E2 26226.715} C_VEL
LIN {X 0,Y 560.279,Z 509.001,A -85,B 0,C 180,E1 26223.464,E2 26223.464} C_VEL
LIN {X 0,Y 560.279,Z 509.225,A -85,B 0,C 180,E1 26222.092,E2 26222.092} C_VEL
LIN {X 0,Y 564.063,Z 520.143,A -85,B 0,C 180,E1 26221.013,E2 26221.013} C_VEL
LIN {X 0,Y 564.292,Z 524.525,A -85,B 0,C 180,E1 26220.682,E2 26220.682} C_VEL
LIN {X 0,Y 563.522,Z 566.616,A -85,B 0,C 180,E1 26217.643,E2 26217.643} C_VEL
LIN {X 0,Y 562.754,Z 612.295,A -85,B 0,C 180,E1 26214.398,E2 26214.398} C_VEL
LIN {X 0,Y 562.867,Z 615.576,A -85,B 0,C 180,E1 26214.215,E2 26214.215} C_VEL
LIN {X 0,Y 563.712,Z 623.031,A -85,B 0,C 180,E1 26214.073,E2 26214.073} C_VEL
LIN {X 0,Y 562.889,Z 824.35,A -85,B 0,C 180,E1 26211.354,E2 26211.354} C_VEL
LIN {X 0,Y 562.643,Z 843.349,A -85,B 0,C 180,E1 26210.904,E2 26210.904} C_VEL
LIN {X 0,Y 562.362,Z 861.413,A -85,B 0,C 180,E1 26210.285,E2 26210.285} C_VEL
LIN {X 0,Y 562.012,Z 879.155,A -85,B 0,C 180,E1 26209.48,E2 26209.48} C_VEL
LIN {X 0,Y 561.664,Z 895.781,A -85,B 0,C 180,E1 26208.527,E2 26208.527} C_VEL
LIN {X 0,Y 561.309,Z 911.633,A -85,B 0,C 180,E1 26207.413,E2 26207.413} C_VEL
LIN {X 0,Y 560.954,Z 926.91,A -85,B 0,C 180,E1 26206.111,E2 26206.111} C_VEL
LIN {X 0,Y 560.642,Z 940.945,A -85,B 0,C 180,E1 26204.67,E2 26204.67} C_VEL
LIN {X 0,Y 560.379,Z 954.087,A -85,B 0,C 180,E1 26203.043,E2 26203.043} C_VEL
LIN {X 0,Y 560.189,Z 964.865,A -85,B 0,C 180,E1 26201.427,E2 26201.427} C_VEL
LIN {X 0,Y 560.056,Z 974.507,A -85,B 0,C 180,E1 26199.661,E2 26199.661} C_VEL
LIN {X 0,Y 559.974,Z 982.176,A -85,B 0,C 180,E1 26197.903,E2 26197.903} C_VEL
LIN {X 0,Y 559.935,Z 988.41,A -85,B 0,C 180,E1 26196.048,E2 26196.048} C_VEL
LIN {X 0,Y 559.921,Z 992.875,A -85,B 0,C 180,E1 26194.2,E2 26194.2} C_VEL
LIN {X 0,Y 559.915,Z 995.79,A -85,B 0,C 180,E1 26192.253,E2 26192.253} C_VEL
LIN {X 0,Y 559.908,Z 996.939,A -85,B 0,C 180,E1 26190.308,E2 26190.308} C_VEL
LIN {X 0,Y 559.913,Z 996.349,A -85,B 0,C 180,E1 26188.364,E2 26188.364} C_VEL
LIN {X 0,Y 559.911,Z 994.006,A -85,B 0,C 180,E1 26186.418,E2 26186.418} C_VEL
LIN {X 0,Y 559.926,Z 990.102,A -85,B 0,C 180,E1 26184.571,E2 26184.571} C_VEL
LIN {X 0,Y 559.956,Z 984.474,A -85,B 0,C 180,E1 26182.718,E2 26182.718} C_VEL
LIN {X 0,Y 560.027,Z 977.435,A -85,B 0,C 180,E1 26180.963,E2 26180.963} C_VEL
LIN {X 0,Y 560.138,Z 968.527,A -85,B 0,C 180,E1 26179.2,E2 26179.2} C_VEL
LIN {X 0,Y 560.309,Z 958.166,A -85,B 0,C 180,E1 26177.533,E2 26177.533} C_VEL
LIN {X 0,Y 560.531,Z 946.369,A -85,B 0,C 180,E1 26175.963,E2 26175.963} C_VEL
LIN {X 0,Y 560.822,Z 932.8,A -85,B 0,C 180,E1 26174.459,E2 26174.459} C_VEL
LIN {X 0,Y 561.16,Z 918.031,A -85,B 0,C 180,E1 26173.099,E2 26173.099} C_VEL
LIN {X 0,Y 561.528,Z 902.273,A -85,B 0,C 180,E1 26171.901,E2 26171.901} C_VEL
LIN {X 0,Y 561.871,Z 885.101,A -85,B 0,C 180,E1 26170.836,E2 26170.836} C_VEL
LIN {X 0,Y 562.252,Z 867.876,A -85,B 0,C 180,E1 26169.985,E2 26169.985} C_VEL
LIN {X 0,Y 562.546,Z 849.626,A -85,B 0,C 180,E1 26169.29,E2 26169.29} C_VEL
LIN {X 0,Y 562.809,Z 831.133,A -85,B 0,C 180,E1 26168.785,E2 26168.785} C_VEL
LIN {X 0,Y 562.977,Z 810.923,A -85,B 0,C 180,E1 26168.441,E2 26168.441} C_VEL
LIN {X 0,Y 563.552,Z 619.962,A -85,B 0,C 180,E1 26165.878,E2 26165.878} C_VEL
LIN {X 0,Y 562.744,Z 614.341,A -85,B 0,C 180,E1 26165.741,E2 26165.741} C_VEL
LIN {X 0,Y 563.494,Z 568.308,A -85,B 0,C 180,E1 26162.479,E2 26162.479} C_VEL
LIN {X 0,Y 564.28,Z 525.377,A -85,B 0,C 180,E1 26159.379,E2 26159.379} C_VEL
LIN {X 0,Y 564.29,Z 520.807,A -85,B 0,C 180,E1 26159.047,E2 26159.047} C_VEL
LIN {X 0,Y 560.293,Z 509.306,A -85,B 0,C 180,E1 26157.928,E2 26157.928} C_VEL
LIN {X 0,Y 560.282,Z 509.004,A -85,B 0,C 180,E1 26156.784,E2 26156.784} C_VEL
LIN {X 0,Y 560.239,Z 509.01,A -85,B 0,C 180,E1 26153.542,E2 26153.542} C_VEL
LIN {X 0,Y 560.283,Z 509.008,A -85,B 0,C 180,E1 26150.277,E2 26150.277} C_VEL
LIN {X 0,Y 560.234,Z 509.007,A -85,B 0,C 180,E1 26147.164,E2 26147.164} C_VEL
LIN {X 0,Y 560.26,Z 509.012,A -85,B 0,C 180,E1 26143.823,E2 26143.823} C_VEL
LIN {X 0,Y 560.251,Z 509.006,A -85,B 0,C 180,E1 26140.647,E2 26140.647} C_VEL
LIN {X 0,Y 560.23,Z 509.01,A -85,B 0,C 180,E1 26137.359,E2 26137.359} C_VEL
LIN {X 0,Y 560.271,Z 509.005,A -85,B 0,C 180,E1 26134.204,E2 26134.204} C_VEL
LIN {X 0,Y 560.218,Z 509.009,A -85,B 0,C 180,E1 26131.051,E2 26131.051} C_VEL
LIN {X 0,Y 560.281,Z 509.006,A -85,B 0,C 180,E1 26127.876,E2 26127.876} C_VEL
LIN {X 0,Y 560.208,Z 509.009,A -85,B 0,C 180,E1 26124.686,E2 26124.686} C_VEL
LIN {X 0,Y 560.264,Z 509.011,A -85,B 0,C 180,E1 26121.46,E2 26121.46} C_VEL
LIN {X 0,Y 560.206,Z 509.008,A -85,B 0,C 180,E1 26118.308,E2 26118.308} C_VEL
LIN {X 0,Y 560.221,Z 509.006,A -85,B 0,C 180,E1 26114.998,E2 26114.998} C_VEL
LIN {X 0,Y 560.204,Z 509.012,A -85,B 0,C 180,E1 26112.049,E2 26112.049} C_VEL
LIN {X 0,Y 560.202,Z 509.01,A -85,B 0,C 180,E1 26108.622,E2 26108.622} C_VEL
LIN {X 0,Y 560.217,Z 509.011,A -85,B 0,C 180,E1 26105.736,E2 26105.736} C_VEL
LIN {X 0,Y 560.21,Z 509.01,A -85,B 0,C 180,E1 26102.455,E2 26102.455} C_VEL
LIN {X 0,Y 560.233,Z 509.008,A -85,B 0,C 180,E1 26099.489,E2 26099.489} C_VEL
LIN {X 0,Y 560.214,Z 509.008,A -85,B 0,C 180,E1 26096.213,E2 26096.213} C_VEL
LIN {X 0,Y 560.275,Z 509.011,A -85,B 0,C 180,E1 26093.03,E2 26093.03} C_VEL
LIN {X 0,Y 560.215,Z 509.007,A -85,B 0,C 180,E1 26089.823,E2 26089.823} C_VEL
LIN {X 0,Y 560.279,Z 509.004,A -85,B 0,C 180,E1 26086.585,E2 26086.585} C_VEL
LIN {X 0,Y 560.228,Z 509.009,A -85,B 0,C 180,E1 26083.395,E2 26083.395} C_VEL
LIN {X 0,Y 560.253,Z 509.005,A -85,B 0,C 180,E1 26080.07,E2 26080.07} C_VEL
LIN {X 0,Y 560.258,Z 509.011,A -85,B 0,C 180,E1 26076.882,E2 26076.882} C_VEL
LIN {X 0,Y 560.28,Z 509.002,A -85,B 0,C 180,E1 26076.214,E2 26076.214} C_VEL
LIN {X 0,Y 559.261,Z 509.128,A -85,B 0,C 180,E1 26075.427,E2 26075.427} C_VEL
LIN {X 0,Y 552.825,Z 509.936,A -85,B 0,C 180,E1 26073.216,E2 26073.216} C_VEL
LIN {X 0,Y 552.334,Z 509.997,A -85,B 0,C 180,E1 26072.64,E2 26072.64} C_VEL
LIN {X 0,Y 552.299,Z 509.997,A -85,B 0,C 180,E1 26069.297,E2 26069.297} C_VEL
LIN {X 0,Y 552.343,Z 509.995,A -85,B 0,C 180,E1 26065.988,E2 26065.988} C_VEL
LIN {X 0,Y 552.322,Z 510,A -85,B 0,C 180,E1 26062.62,E2 26062.62} C_VEL
LIN {X 0,Y 552.313,Z 510.002,A -85,B 0,C 180,E1 26059.192,E2 26059.192} C_VEL
LIN {X 0,Y 552.367,Z 510.29,A -85,B 0,C 180,E1 26058.531,E2 26058.531} C_VEL
LIN {X 0,Y 554.972,Z 520.347,A -85,B 0,C 180,E1 26057.154,E2 26057.154} C_VEL
LIN {X 0,Y 554.182,Z 548.616,A -85,B 0,C 180,E1 26053.806,E2 26053.806} C_VEL
LIN {X 0,Y 553.539,Z 577.943,A -85,B 0,C 180,E1 26050.42,E2 26050.42} C_VEL
LIN {X 0,Y 553.036,Z 609.015,A -85,B 0,C 180,E1 26046.954,E2 26046.954} C_VEL
LIN {X 0,Y 552.723,Z 632.961,A -85,B 0,C 180,E1 26044.356,E2 26044.356} C_VEL
LIN {X 0,Y 553.457,Z 640.751,A -85,B 0,C 180,E1 26044.218,E2 26044.218} C_VEL
LIN {X 0,Y 553.121,Z 744.379,A -85,B 0,C 180,E1 26042.843,E2 26042.843} C_VEL
LIN {X 0,Y 553.033,Z 758.682,A -85,B 0,C 180,E1 26042.472,E2 26042.472} C_VEL
LIN {X 0,Y 552.861,Z 772.935,A -85,B 0,C 180,E1 26041.902,E2 26041.902} C_VEL
LIN {X 0,Y 552.645,Z 786.482,A -85,B 0,C 180,E1 26041.155,E2 26041.155} C_VEL
LIN {X 0,Y 552.439,Z 799.191,A -85,B 0,C 180,E1 26040.232,E2 26040.232} C_VEL
LIN {X 0,Y 552.271,Z 810.792,A -85,B 0,C 180,E1 26039.14,E2 26039.14} C_VEL
LIN {X 0,Y 552.129,Z 820.606,A -85,B 0,C 180,E1 26037.967,E2 26037.967} C_VEL
LIN {X 0,Y 552.021,Z 829.022,A -85,B 0,C 180,E1 26036.688,E2 26036.688} C_VEL
LIN {X 0,Y 551.958,Z 836.439,A -85,B 0,C 180,E1 26035.191,E2 26035.191} C_VEL
LIN {X 0,Y 551.928,Z 841.655,A -85,B 0,C 180,E1 26033.71,E2 26033.71} C_VEL
LIN {X 0,Y 551.919,Z 845.082,A -85,B 0,C 180,E1 26032.22,E2 26032.22} C_VEL
LIN {X 0,Y 551.919,Z 846.855,A -85,B 0,C 180,E1 26030.573,E2 26030.573} C_VEL
LIN {X 0,Y 551.915,Z 846.622,A -85,B 0,C 180,E1 26028.973,E2 26028.973} C_VEL
LIN {X 0,Y 551.919,Z 844.735,A -85,B 0,C 180,E1 26027.498,E2 26027.498} C_VEL
LIN {X 0,Y 551.931,Z 841.017,A -85,B 0,C 180,E1 26025.981,E2 26025.981} C_VEL
LIN {X 0,Y 551.961,Z 835.832,A -85,B 0,C 180,E1 26024.581,E2 26024.581} C_VEL
LIN {X 0,Y 552.021,Z 828.838,A -85,B 0,C 180,E1 26023.19,E2 26023.19} C_VEL
LIN {X 0,Y 552.141,Z 819.589,A -85,B 0,C 180,E1 26021.805,E2 26021.805} C_VEL
LIN {X 0,Y 552.291,Z 809.54,A -85,B 0,C 180,E1 26020.639,E2 26020.639} C_VEL
LIN {X 0,Y 552.469,Z 798,A -85,B 0,C 180,E1 26019.582,E2 26019.582} C_VEL
LIN {X 0,Y 552.669,Z 785.422,A -85,B 0,C 180,E1 26018.687,E2 26018.687} C_VEL
LIN {X 0,Y 552.879,Z 771.706,A -85,B 0,C 180,E1 26017.95,E2 26017.95} C_VEL
LIN {X 0,Y 553.049,Z 757.529,A -85,B 0,C 180,E1 26017.402,E2 26017.402} C_VEL
LIN {X 0,Y 553.173,Z 742.245,A -85,B 0,C 180,E1 26017.026,E2 26017.026} C_VEL
LIN {X 0,Y 553.23,Z 636.593,A -85,B 0,C 180,E1 26015.631,E2 26015.631} C_VEL
LIN {X 0,Y 552.761,Z 632.899,A -85,B 0,C 180,E1 26015.552,E2 26015.552} C_VEL
LIN {X 0,Y 553.085,Z 602.905,A -85,B 0,C 180,E1 26012.278,E2 26012.278} C_VEL
LIN {X 0,Y 553.624,Z 572.399,A -85,B 0,C 180,E1 26008.861,E2 26008.861} C_VEL
LIN {X 0,Y 554.242,Z 543.685,A -85,B 0,C 180,E1 26005.55,E2 26005.55} C_VEL
LIN {X 0,Y 554.854,Z 519.955,A -85,B 0,C 180,E1 26002.753,E2 26002.753} C_VEL
LIN {X 0,Y 552.319,Z 510.083,A -85,B 0,C 180,E1 26001.358,E2 26001.358} C_VEL
LIN {X 0,Y 552.269,Z 510.003,A -85,B 0,C 180,E1 25998.301,E2 25998.301} C_VEL
LIN {X 0,Y 552.276,Z 510.001,A -85,B 0,C 180,E1 25994.888,E2 25994.888} C_VEL
LIN {X 0,Y 552.281,Z 510,A -85,B 0,C 180,E1 25991.857,E2 25991.857} C_VEL
LIN {X 0,Y 552.263,Z 510,A -85,B 0,C 180,E1 25988.527,E2 25988.527} C_VEL
LIN {X 0,Y 552.294,Z 509.987,A -85,B 0,C 180,E1 25985.508,E2 25985.508} C_VEL
LIN {X 0,Y 552.258,Z 510,A -85,B 0,C 180,E1 25982.272,E2 25982.272} C_VEL
LIN {X 0,Y 552.318,Z 509.985,A -85,B 0,C 180,E1 25979.102,E2 25979.102} C_VEL
LIN {X 0,Y 552.254,Z 510,A -85,B 0,C 180,E1 25975.859,E2 25975.859} C_VEL
LIN {X 0,Y 552.318,Z 509.998,A -85,B 0,C 180,E1 25972.629,E2 25972.629} C_VEL
LIN {X 0,Y 552.257,Z 510,A -85,B 0,C 180,E1 25969.6,E2 25969.6} C_VEL
LIN {X 0,Y 552.318,Z 509.998,A -85,B 0,C 180,E1 25966.395,E2 25966.395} C_VEL
LIN {X 0,Y 552.263,Z 510,A -85,B 0,C 180,E1 25963.3,E2 25963.3} C_VEL
LIN {X 0,Y 552.295,Z 509.997,A -85,B 0,C 180,E1 25959.993,E2 25959.993} C_VEL
LIN {X 0,Y 552.27,Z 510,A -85,B 0,C 180,E1 25957.026,E2 25957.026} C_VEL
LIN {X 0,Y 552.281,Z 509.993,A -85,B 0,C 180,E1 25953.619,E2 25953.619} C_VEL
LIN {X 0,Y 552.29,Z 509.999,A -85,B 0,C 180,E1 25950.579,E2 25950.579} C_VEL
LIN {X 0,Y 552.274,Z 509.993,A -85,B 0,C 180,E1 25947.261,E2 25947.261} C_VEL
LIN {X 0,Y 552.32,Z 509.994,A -85,B 0,C 180,E1 25944.15,E2 25944.15} C_VEL
LIN {X 0,Y 552.272,Z 509.997,A -85,B 0,C 180,E1 25940.895,E2 25940.895} C_VEL
LIN {X 0,Y 552.341,Z 509.989,A -85,B 0,C 180,E1 25937.705,E2 25937.705} C_VEL
LIN {X 0,Y 552.274,Z 509.997,A -85,B 0,C 180,E1 25934.576,E2 25934.576} C_VEL
LIN {X 0,Y 552.338,Z 509.992,A -85,B 0,C 180,E1 25931.38,E2 25931.38} C_VEL
LIN {X 0,Y 552.279,Z 509.989,A -85,B 0,C 180,E1 25928.223,E2 25928.223} C_VEL
LIN {X 0,Y 552.308,Z 509.995,A -85,B 0,C 180,E1 25924.881,E2 25924.881} C_VEL
LIN {X 0,Y 552.297,Z 509.996,A -85,B 0,C 180,E1 25921.764,E2 25921.764} C_VEL
LIN {X 0,Y 552.286,Z 509.994,A -85,B 0,C 180,E1 25918.34,E2 25918.34} C_VEL
LIN {X 0,Y 552.341,Z 509.997,A -85,B 0,C 180,E1 25915.12,E2 25915.12} C_VEL
LIN {X 0,Y 552.284,Z 509.99,A -85,B 0,C 180,E1 25911.882,E2 25911.882} C_VEL
LIN {X 0,Y 552.339,Z 509.994,A -85,B 0,C 180,E1 25908.62,E2 25908.62} C_VEL
LIN {X 0,Y 552.294,Z 509.993,A -85,B 0,C 180,E1 25905.425,E2 25905.425} C_VEL
LIN {X 0,Y 552.3,Z 509.995,A -85,B 0,C 180,E1 25901.967,E2 25901.967} C_VEL
LIN {X 0,Y 552.334,Z 509.994,A -85,B 0,C 180,E1 25898.774,E2 25898.774} C_VEL
LIN {X 0,Y 552.292,Z 509.996,A -85,B 0,C 180,E1 25895.507,E2 25895.507} C_VEL
LIN {X 0,Y 552.346,Z 509.995,A -85,B 0,C 180,E1 25892.268,E2 25892.268} C_VEL
LIN {X 0,Y 552.298,Z 509.995,A -85,B 0,C 180,E1 25889.06,E2 25889.06} C_VEL
LIN {X 0,Y 552.328,Z 509.992,A -85,B 0,C 180,E1 25885.737,E2 25885.737} C_VEL
LIN {X 0,Y 552.331,Z 509.999,A -85,B 0,C 180,E1 25882.407,E2 25882.407} C_VEL
LIN {X 0,Y 552.301,Z 509.996,A -85,B 0,C 180,E1 25879.054,E2 25879.054} C_VEL
LIN {X 0,Y 552.342,Z 509.993,A -85,B 0,C 180,E1 25875.791,E2 25875.791} C_VEL
LIN {X 0,Y 552.305,Z 509.998,A -85,B 0,C 180,E1 25872.471,E2 25872.471} C_VEL
LIN {X 0,Y 552.321,Z 509.994,A -85,B 0,C 180,E1 25869.046,E2 25869.046} C_VEL
LIN {X 0,Y 552.34,Z 510,A -85,B 0,C 180,E1 25865.78,E2 25865.78} C_VEL
LIN {X 0,Y 552.326,Z 510.149,A -85,B 0,C 180,E1 25862.509,E2 25862.509} C_VEL
LIN {X 0,Y 553.966,Z 515.115,A -85,B 0,C 180,E1 25861.972,E2 25861.972} C_VEL
LIN {X 0,Y 556.964,Z 524.249,A -85,B 0,C 180,E1 25861.096,E2 25861.096} C_VEL
LIN {X 0,Y 556.188,Z 567.403,A -85,B 0,C 180,E1 25857.981,E2 25857.981} C_VEL
LIN {X 0,Y 555.288,Z 612.295,A -85,B 0,C 180,E1 25854.748,E2 25854.748} C_VEL
LIN {X 0,Y 555.386,Z 615.535,A -85,B 0,C 180,E1 25854.563,E2 25854.563} C_VEL
LIN {X 0,Y 556.404,Z 623.852,A -85,B 0,C 180,E1 25854.398,E2 25854.398} C_VEL
LIN {X 0,Y 555.436,Z 824.349,A -85,B 0,C 180,E1 25851.655,E2 25851.655} C_VEL
LIN {X 0,Y 555.153,Z 843.307,A -85,B 0,C 180,E1 25851.201,E2 25851.201} C_VEL
LIN {X 0,Y 554.818,Z 861.411,A -85,B 0,C 180,E1 25850.573,E2 25850.573} C_VEL
LIN {X 0,Y 554.413,Z 879.052,A -85,B 0,C 180,E1 25849.764,E2 25849.764} C_VEL
LIN {X 0,Y 553.991,Z 895.792,A -85,B 0,C 180,E1 25848.792,E2 25848.792} C_VEL
LIN {X 0,Y 553.575,Z 911.631,A -85,B 0,C 180,E1 25847.664,E2 25847.664} C_VEL
LIN {X 0,Y 553.164,Z 926.559,A -85,B 0,C 180,E1 25846.378,E2 25846.378} C_VEL
LIN {X 0,Y 552.809,Z 940.019,A -85,B 0,C 180,E1 25844.989,E2 25844.989} C_VEL
LIN {X 0,Y 552.497,Z 952.913,A -85,B 0,C 180,E1 25843.394,E2 25843.394} C_VEL
LIN {X 0,Y 552.263,Z 964.229,A -85,B 0,C 180,E1 25841.699,E2 25841.699} C_VEL
LIN {X 0,Y 552.095,Z 974.172,A -85,B 0,C 180,E1 25839.87,E2 25839.87} C_VEL
LIN {X 0,Y 551.988,Z 982.175,A -85,B 0,C 180,E1 25838.018,E2 25838.018} C_VEL
LIN {X 0,Y 551.941,Z 988.41,A -85,B 0,C 180,E1 25836.136,E2 25836.136} C_VEL
LIN {X 0,Y 551.921,Z 992.875,A -85,B 0,C 180,E1 25834.26,E2 25834.26} C_VEL
LIN {X 0,Y 551.915,Z 995.791,A -85,B 0,C 180,E1 25832.285,E2 25832.285} C_VEL
LIN {X 0,Y 551.908,Z 996.939,A -85,B 0,C 180,E1 25830.313,E2 25830.313} C_VEL
LIN {X 0,Y 551.913,Z 996.348,A -85,B 0,C 180,E1 25828.34,E2 25828.34} C_VEL
LIN {X 0,Y 551.913,Z 994.005,A -85,B 0,C 180,E1 25826.366,E2 25826.366} C_VEL
LIN {X 0,Y 551.928,Z 990.102,A -85,B 0,C 180,E1 25824.492,E2 25824.492} C_VEL
LIN {X 0,Y 551.968,Z 984.474,A -85,B 0,C 180,E1 25822.613,E2 25822.613} C_VEL
LIN {X 0,Y 552.055,Z 977.212,A -85,B 0,C 180,E1 25820.78,E2 25820.78} C_VEL
LIN {X 0,Y 552.186,Z 968.528,A -85,B 0,C 180,E1 25819.042,E2 25819.042} C_VEL
LIN {X 0,Y 552.392,Z 957.973,A -85,B 0,C 180,E1 25817.322,E2 25817.322} C_VEL
LIN {X 0,Y 552.654,Z 946.37,A -85,B 0,C 180,E1 25815.759,E2 25815.759} C_VEL
LIN {X 0,Y 553.007,Z 932.6,A -85,B 0,C 180,E1 25814.213,E2 25814.213} C_VEL
LIN {X 0,Y 553.414,Z 917.636,A -85,B 0,C 180,E1 25812.822,E2 25812.822} C_VEL
LIN {X 0,Y 553.852,Z 901.476,A -85,B 0,C 180,E1 25811.586,E2 25811.586} C_VEL
LIN {X 0,Y 554.246,Z 885.103,A -85,B 0,C 180,E1 25810.562,E2 25810.562} C_VEL
LIN {X 0,Y 554.685,Z 867.878,A -85,B 0,C 180,E1 25809.7,E2 25809.7} C_VEL
LIN {X 0,Y 555.036,Z 849.629,A -85,B 0,C 180,E1 25808.996,E2 25808.996} C_VEL
LIN {X 0,Y 555.345,Z 830.968,A -85,B 0,C 180,E1 25808.483,E2 25808.483} C_VEL
LIN {X 0,Y 555.539,Z 810.606,A -85,B 0,C 180,E1 25808.133,E2 25808.133} C_VEL
LIN {X 0,Y 556.24,Z 620.997,A -85,B 0,C 180,E1 25805.554,E2 25805.554} C_VEL
LIN {X 0,Y 555.27,Z 614.432,A -85,B 0,C 180,E1 25805.399,E2 25805.399} C_VEL
LIN {X 0,Y 556.156,Z 569.017,A -85,B 0,C 180,E1 25802.137,E2 25802.137} C_VEL
LIN {X 0,Y 556.945,Z 525.438,A -85,B 0,C 180,E1 25798.991,E2 25798.991} C_VEL
LIN {X 0,Y 556.863,Z 523.344,A -85,B 0,C 180,E1 25798.832,E2 25798.832} C_VEL
LIN {X 0,Y 552.338,Z 510.238,A -85,B 0,C 180,E1 25797.519,E2 25797.519} C_VEL
LIN {X 0,Y 552.342,Z 509.997,A -85,B 0,C 180,E1 25794.351,E2 25794.351} C_VEL
LIN {X 0,Y 552.308,Z 509.995,A -85,B 0,C 180,E1 25791.089,E2 25791.089} C_VEL
LIN {X 0,Y 552.304,Z 509.998,A -85,B 0,C 180,E1 25787.673,E2 25787.673} C_VEL
LIN {X 0,Y 552.341,Z 509.995,A -85,B 0,C 180,E1 25784.471,E2 25784.471} C_VEL
LIN {X 0,Y 552.288,Z 509.997,A -85,B 0,C 180,E1 25781.146,E2 25781.146} C_VEL
LIN {X 0,Y 552.335,Z 509.999,A -85,B 0,C 180,E1 25777.855,E2 25777.855} C_VEL
LIN {X 0,Y 552.29,Z 509.996,A -85,B 0,C 180,E1 25774.643,E2 25774.643} C_VEL
LIN {X 0,Y 552.283,Z 509.999,A -85,B 0,C 180,E1 25771.183,E2 25771.183} C_VEL
LIN {X 0,Y 552.322,Z 509.995,A -85,B 0,C 180,E1 25768.078,E2 25768.078} C_VEL
LIN {X 0,Y 552.271,Z 509.998,A -85,B 0,C 180,E1 25764.836,E2 25764.836} C_VEL
LIN {X 0,Y 552.342,Z 509.998,A -85,B 0,C 180,E1 25761.671,E2 25761.671} C_VEL
LIN {X 0,Y 552.263,Z 509.997,A -85,B 0,C 180,E1 25758.453,E2 25758.453} C_VEL
LIN {X 0,Y 552.305,Z 509.995,A -85,B 0,C 180,E1 25755.218,E2 25755.218} C_VEL
LIN {X 0,Y 552.262,Z 510.001,A -85,B 0,C 180,E1 25752.123,E2 25752.123} C_VEL
LIN {X 0,Y 552.271,Z 509.999,A -85,B 0,C 180,E1 25748.737,E2 25748.737} C_VEL
LIN {X 0,Y 552.272,Z 510,A -85,B 0,C 180,E1 25745.819,E2 25745.819} C_VEL
LIN {X 0,Y 552.269,Z 509.999,A -85,B 0,C 180,E1 25742.386,E2 25742.386} C_VEL
LIN {X 0,Y 552.319,Z 509.995,A -85,B 0,C 180,E1 25739.274,E2 25739.274} C_VEL
